(* CODESYS project CtaAppAbtauung_1.0.0.1.library
   Description: Abtauungs Library der CTA
   Version: 1.0.0.1
   Title: CtaAppAbtauung
   Author: SIS
   DocFormat: reStructuredText
   LanguageModelAttribute: qualified-access-only
   Placeholder: CtaAppAbtauung
   CompiledLibraryCompatibilityVersion: CODESYS V3.5 SP16 Patch 3
   Company: CTA
   DefaultNamespace: CtaAppAbtauung

Project tree, tasks and I/O mapping:
  libraries: CtaSysConfig, 1.0.0.2 (CTA); VisuSymbols, 4.5.0.0 (System); CtaVisSymbols, 1.0.0.1 (CTA); Standard, 3.5.18.0 (System); CtaAppInfluxLog, 1.0.0.1 (CTA); CtaVisApps, 1.0.0.0 (CTA); CtaVisHelp, 1.0.0.0 (CTA); CtaVisUser, 1.0.0.0 (CTA); WagoSysVisuBACnet, 2.0.0.0 (WAGO); WagoVisuIcons, 1.1.0.5 (WAGO); WagoVisuIconsMaterialDesign, 1.0.0.0 (WAGO); CtaAppBasic, 1.0.0.1 (CTA); CtaAppReport, 1.0.0.2 (CTA); CtaAppBmk, 1.0.0.0 (CTA); CtaAppTime, 1.0.0.1 (CTA)
  40 Visualizations/
    DIALOG/
      visualisation DIA_ParameterAbtauung
      visualisation DIA_Aussentemperatur
      visualisation DIA_Abtauukriterium
      visualisation DIA_Abtauuanforderung
    ICON/
      visualisation VIS_ABTAUUNG
      visualisation VIS_ABTAUUNG_CheckQuerry
      visualisation VIS_ABTAUUNG_OPEN
    visualisation VIS_AbtauungInfo
    visualisation VIS_AbtauungInfoQuerry
  30 Program Organization Units/
    function block fbAbtauung [ST]: actConfig, actTrendlog, actReport, actState, proAcknowledge, proAvailable, proLockDown, proIsError, proIsWarning, proConfigError, p_scAbtauungHilfsenergie_fbiRepTilLockdown, p_scAbtauungHilfsenergie_fbrTempAbtauEnde, p_scAbtauungHilfsenergie_fbtMaxAbtauungHiEnergie, p_scAbtauungHilfsenergie_fbudiAbtauungenHiEnergie, p_scAbtropfphase_fbtAbtropfzeit, p_scBase_fbtAbtauverzögerung, p_scBase_fbtSperrungAbtauung, p_scBase_fbrAtfürAbtauusperre, p_scManual_fbuiManualState, p_scManual_fbxManualResetLockTime, p_scUmluftabtauung_fbrTempAbtauUmluftOk, p_scUmluftabtauung_fbtAbtauzeitUmluft, p_scUmluftabtauung_fbudiAbtauungenUmluft, p_scAbtauukriterium_fbrAbtauukriteriumFix, p_scAbtauukriterium_fbrKorrekturAtLuftkühler, p_scTable_fbr_dT_Leistung1, p_scTable_fbr_dT_Leistung2, p_scTable_fbr_dT_LeistungMax, p_scTable_fbr_dT_LeistungMin, p_scTable_fbrAtLeistung1, p_scTable_fbrAtLeistung2, p_scTable_fbrAtLeistungMax, p_scTable_fbrAtLeistungMin, p_scTable_fbrAtMaxLeistung1, p_scTable_fbrAtMaxLeistung2, p_scTable_fbrAtMaxLeistungMax, p_scTable_fbrAtMaxLeistungMin, p_scTable_fbrAtMinLeistung1, p_scTable_fbrAtMinLeistung2, p_scTable_fbrAtMinLeistungMax, p_scTable_fbrAtMinLeistungMin, p_scTable_fbrAussenaemperaturMax, p_scTable_fbrAussentemperatur, p_scTable_fbrAussentemperaturMin, p_scTable_fbrLeistung1, p_scTable_fbrLeistung2, p_scTable_fbrMaxLeistung, p_scTable_fbrMinLeistung, p_scAussentemperatur_fbtAverageTimeRange, p_scAussentemperatur_fbxAtGemittelt, p_scInfluxDb_fbxEnable, proITF_REPORTMANAGER, prorActAussentemperatur, prorActAustrittstemperatur, prorZieltemperatur, prorActdTAbtauukriterium, prorAbtaukriteriumFix, prorKorrekturfaktorRk, prorActdTRückkühler, prordTAuslegung, prordTLeistung, proxSperrungAktiv, proudiActHilfsenergieAbtauungen, proudiActUmluftAbtaaungen, protSperrzeit, protStartverzögerung, proiStatus, proxAcknowledge, proxDemandAbtauung, proxDemandManualAbtauung, proxGenerelleDemand, proxDemandHilfsenergie, proManualUmluft, proManualHilfsenergie, proManualBeenden, proManualQuitTime, protTimeLeftAbtropfen, protTimeLeftUmluft, protTimeLeftHilfsenergie, protElapsedUmluft, protElapsedHilfsenergie
  00000000-0000-0000-0000-000000000000|D:\CoDeSys\LibrariesV3\trunk\Intern\CAA\CAA Template\3.4.0.0 draft\Placeholder.xml
  00000000-0000-0000-0000-000000000000|D:\CoDeSys\LibrariesV3\trunk\Intern\CAA\CAA Template\3.2.0.3 draft\Prefix.pdf
  00000000-0000-0000-0000-000000000000|D:\CoDeSys\LibrariesV3\trunk\Intern\CAA\CAA Template\3.5.2.0 draft\Placeholder.xml
  20 Structs/
    data type scParameter
    Abtauukriterium/
      Tabelle/
        data type scTable
      data type scAbtauukriterium
    Abtauuanforderung/
      data type scAbtauuanforderung
      Base/
        data type scBase
      Umluftabtauung/
        data type scUmluftabtauung
      AbtauungHilfsenergie/
        data type scAbtauungHilfsenergie
      Abtropfphase/
        data type scAbtropfphase
      Manual/
        data type scManual
    Aussentemperatur/
      data type scAussentemperatur
    Trend/
      data type scTrend
    InfluxDb/
      data type scInfluxDb
  50 Images/
  10 Documenation/
    global variables VersionHistory
    global variables readMe
  21 Interface/
    interface ITF_Abtauung: proAcknowledge, proAvailable, proLockDown, proIsError, proIsWarning, prorActdTAbtauukriterium, prorKorrekturfaktorRk, prorAbtaukriteriumFix, prorActAustrittstemperatur, prorActAussentemperatur, prorZieltemperatur, proxDemandAbtauung, proxDemandManualAbtauung, proxGenerelleDemand, proxDemandHilfsenergie, proxSperrungAktiv, proudiActUmluftAbtaaungen, proudiActHilfsenergieAbtauungen, protSperrzeit, protStartverzögerung, proiStatus, proxAcknowledge, prordTAuslegung, prordTLeistung, prorActdTRückkühler, protTimeLeftAbtropfen, protTimeLeftUmluft, protTimeLeftHilfsenergie, protElapsedUmluft, protElapsedHilfsenergie, p_scAbtauungHilfsenergie_fbudiAbtauungenHiEnergie, p_scAbtauungHilfsenergie_fbrTempAbtauEnde, p_scAbtauungHilfsenergie_fbtMaxAbtauungHiEnergie, p_scAbtauungHilfsenergie_fbiRepTilLockdown, p_scAbtropfphase_fbtAbtropfzeit, p_scBase_fbtAbtauverzögerung, p_scBase_fbtSperrungAbtauung, p_scBase_fbrAtfürAbtauusperre, p_scManual_fbxManualResetLockTime, p_scManual_fbuiManualState, p_scUmluftabtauung_fbrTempAbtauUmluftOk, p_scUmluftabtauung_fbtAbtauzeitUmluft, p_scUmluftabtauung_fbudiAbtauungenUmluft, p_scInfluxDb_fbxEnable, p_scAbtauukriterium_fbrAbtauukriteriumFix, p_scAbtauukriterium_fbrKorrekturAtLuftkühler, p_scTable_fbrAtLeistungMax, p_scTable_fbrAtMinLeistung1, p_scTable_fbr_dT_LeistungMin, p_scTable_fbrAtMaxLeistungMax, p_scTable_fbrAtMaxLeistung1, p_scTable_fbr_dT_Leistung2, p_scTable_fbr_dT_Leistung1, p_scTable_fbrAtMaxLeistung2, p_scTable_fbrAussenaemperaturMax, p_scTable_fbrAussentemperaturMin, p_scTable_fbrLeistung2, p_scTable_fbrMinLeistung, p_scTable_fbrAtMinLeistungMax, p_scTable_fbrAtLeistung1, p_scTable_fbrLeistung1, p_scTable_fbrMaxLeistung, p_scTable_fbrAussentemperatur, p_scTable_fbrAtMinLeistungMin, p_scTable_fbrAtMinLeistung2, p_scTable_fbrAtMaxLeistungMin, p_scTable_fbrAtLeistungMin, p_scTable_fbrAtLeistung2, p_scTable_fbr_dT_LeistungMax, p_scAussentemperatur_fbtAverageTimeRange, p_scAussentemperatur_fbxAtGemittelt, proConfigError, proITF_REPORTMANAGER, proManualUmluft, proManualHilfsenergie, proManualBeenden, proManualQuitTime
  11 Library Parameter/
  12 Konstanten/
  60 Textlisten/
    text list Error
    text list Info
    text list Warnung
  13 Globale Variablen/
    global variables GlobalKonstant
  text list GlobalTextList
*)

// 20 Structs/scParameter
TYPE scParameter :
    STRUCT
	// Parameter
	scAbtauuanforderung		:	scAbtauuanforderung;
	scAussentemperatur		:	scAussentemperatur;
	scAbtauukriterium		:	scAbtauukriterium;
	scInfluxDb				:	scInfluxDb;
	scTrend					:	scTrend;
    END_STRUCT
END_TYPE

// 20 Structs/Abtauukriterium/Tabelle/scTable
TYPE scTable :
	STRUCT
		(*Leistungen*)
		fbrMinLeistung				:	CtaSysConfig.fbREAL;
		fbrLeistung1				:	CtaSysConfig.fbREAL;
		fbrLeistung2				:	CtaSysConfig.fbREAL;
		fbrMaxLeistung				:	CtaSysConfig.fbREAL;
		(*Aussentemperaturen*)
		fbrAussentemperaturMin		:	CtaSysConfig.fbREAL;
		fbrAussentemperatur			:	CtaSysConfig.fbREAL;
		fbrAussenaemperaturMax		:	CtaSysConfig.fbREAL;
		(*dT*)
		fbrAtMinLeistungMin			:	CtaSysConfig.fbREAL;
		fbrAtMinLeistung1			:	CtaSysConfig.fbREAL;
		fbrAtMinLeistung2			:	CtaSysConfig.fbREAL;
		fbrAtMinLeistungMax			:	CtaSysConfig.fbREAL;		
		fbrAtLeistungMin			:	CtaSysConfig.fbREAL;
		fbrAtLeistung1				:	CtaSysConfig.fbREAL;
		fbrAtLeistung2				:	CtaSysConfig.fbREAL;
		fbrAtLeistungMax			:	CtaSysConfig.fbREAL;		
		fbrAtMaxLeistungMin			:	CtaSysConfig.fbREAL;
		fbrAtMaxLeistung1			:	CtaSysConfig.fbREAL;
		fbrAtMaxLeistung2			:	CtaSysConfig.fbREAL;
		fbrAtMaxLeistungMax			:	CtaSysConfig.fbREAL;
		(*dT's für Auslösungen*)
		fbr_dT_LeistungMin			:	CtaSysConfig.fbREAL;
		fbr_dT_Leistung1			:	CtaSysConfig.fbREAL;
		fbr_dT_Leistung2			:	CtaSysConfig.fbREAL;
		fbr_dT_LeistungMax			:	CtaSysConfig.fbREAL;
	END_STRUCT
END_TYPE

// 20 Structs/Abtauukriterium/scAbtauukriterium
TYPE scAbtauukriterium :
	STRUCT
		scTable 					:	scTable;
		fbrKorrekturAtLuftkühler	:	CtaSysConfig.fbREAL;		
		fbrAbtauukriteriumFix		:	CtaSysConfig.fbREAL;
	END_STRUCT
END_TYPE

// 20 Structs/Abtauuanforderung/scAbtauuanforderung
TYPE scAbtauuanforderung :
	STRUCT
		scBase					:	scBase;
		scUmluftabtauung		:	scUmluftabtauung;
		scAbtauungHilfsenergie	:	scAbtauungHilfsenergie;
		scAbtropfphase			:	scAbtropfphase;
		scManual				:	scManual;		
	END_STRUCT
END_TYPE

// 20 Structs/Aussentemperatur/scAussentemperatur
TYPE scAussentemperatur :
	STRUCT
		fbxAtGemittelt				:	CtaSysConfig.fbBOOL;
		fbtAverageTimeRange			:	CtaSysConfig.fbTIME;		
	END_STRUCT
END_TYPE

// 20 Structs/Abtauuanforderung/AbtauungHilfsenergie/scAbtauungHilfsenergie
TYPE scAbtauungHilfsenergie :
	STRUCT
		fbrTempAbtauEnde			:	CtaSysConfig.fbREAL;
		fbtMaxAbtauungHiEnergie		:	CtaSysConfig.fbTIME;
		fbiRepTilLockdown			:	CtaSysConfig.fbINT;
		fbudiAbtauungenHiEnergie	:	CtaSysConfig.fbUDINT;
	END_STRUCT
END_TYPE

// 20 Structs/Abtauuanforderung/Abtropfphase/scAbtropfphase
TYPE scAbtropfphase :
	STRUCT
		fbtAbtropfzeit				:	CtaSysConfig.fbTIME;	
	END_STRUCT
END_TYPE

// 20 Structs/Abtauuanforderung/Base/scBase
TYPE scBase :
	STRUCT
		fbtAbtauverzögerung			:	CtaSysConfig.fbTIME;
		fbtSperrungAbtauung			:	CtaSysConfig.fbTIME;
		fbrAtfürAbtauusperre		:	CtaSysConfig.fbREAL;
	END_STRUCT
END_TYPE

// 20 Structs/Abtauuanforderung/Manual/scManual
TYPE scManual :
	STRUCT
		fbxManualResetLockTime	:	CtaSysConfig.fbBOOL;	// Manuelle rücksetzung der Sperrzeit
		fbuiManualState			:	CtaSysConfig.fbUINT;	// 0 = Off, 1 = Umluftabtauung, 2 = Abtauung mit Hilfsenergie , 3 = Abtauung Beenden
	END_STRUCT
END_TYPE

// 20 Structs/Abtauuanforderung/Umluftabtauung/scUmluftabtauung
TYPE scUmluftabtauung :
	STRUCT
		fbrTempAbtauUmluftOk		:	CtaSysConfig.fbREAL;
		fbtAbtauzeitUmluft			:	CtaSysConfig.fbTIME;	
		fbudiAbtauungenUmluft		:	CtaSysConfig.fbUDINT;
	END_STRUCT
END_TYPE

// 20 Structs/Trend/scTrend
TYPE scTrend :
	STRUCT
		fbxEnable	: CtaSysConfig.fbBOOL;
	END_STRUCT
END_TYPE

// 20 Structs/InfluxDb/scInfluxDb
{attribute 'pack_mode' := '1'} 
TYPE scInfluxDb :
    STRUCT
        fbxEnable       :   CtaSysConfig.fbBOOL;
    END_STRUCT
END_TYPE

// 10 Documenation/VersionHistory
(* 

.. image:: ../../Images/CTA_Logo.jpg
   :align: right
   :width: 15% 

**Vorlage**   


============ =========== =========== ============================================
**Date**     **Version** **Author**  **Change**
------------ ----------- ----------- --------------------------------------------
04.03.2021   0.0.0.0     SIS         Vorlage erstellt

============ =========== =========== ============================================


*)
VAR_GLOBAL
    stInfo : STRING:= '0.0.0.0, Vorlage, CTA';
END_VAR

// 10 Documenation/readMe
(*

**ReadMe**
 
 |  **Empfehlung**
 |
 |	Bibliothek CtaAppPid zur implementierung eine PID- Reglers.
 |  Instanzieren Sie den CtaAppPid.fbPid in ihrem Funktionsbaustein oder POU beispielsweise als fbPidX(Komponente)Y. (X = Nr des Reglers; Komponente z.B Pumpe, Antrieb oder Ventilator; Y = Nr der Komponente) 
 |  Deklarieren Sie die Struktur Variable welche als Parameter und zur ansteuerung dienen wie im Code beispiel.
 |  
 |  *Beispiel* 

+-----------------------+---------------------------------------------------------------------------------------------------------------------------------------------------------------------------------------------------------------------------------------------------------------------------------------------------------------------------------------------------------------------------------------------------------------------------------------+
| Beschreibung          |  Code                                                                                                                                                                                                                                                                                                                                                                                                                                 |
+=======================+=======================================================================================================================================================================================================================================================================================================================================================================================================================================+
| Pou oder SmFb         | .. code-block:: codesys                                                                                                                                                                                                                                                                                                                                                                                                               |
|                       |                                                                                                                                                                                                                                                                                                                                                                                                                                       |
|                       |	// Deklaration als VAR im POU oder dem selbsterstellten Funktionsbaustein                                                                                                                                                                                                                                                                                                                                                       	|
|                       |   VAR   																																																																																																								|
|						|	    (*PID*)																																																	 																																																						|
|						|		fbPid1Pumpe1			: CtaAppPid.fbPid;                                                                                                                                                                                                                                                                                                                                                              						|
|                       | 		fbPid2Pumpe1			: CtaAppPid.fbPid;																																																																																														|
| 						|	END_VAR                                                                                                                                                                                                                                                                                                                                                                                                                         	|
+-----------------------+---------------------------------------------------------------------------------------------------------------------------------------------------------------------------------------------------------------------------------------------------------------------------------------------------------------------------------------------------------------------------------------------------------------------------------------+
| Code für Init         | .. code-block:: codesys                                                                                                                                                                                                                                                                                                                                                                                                               |
|                       |   																																																																																																									|
| 						|	// Kopieren des nachfolgenden Codes in eine Action zur Initialisierung der Parameter. Zum Beispiel actParameter.																																																																													|
|                       |	{region "Parameter Pid1Pumpe1"}                                                                                                                                                                                                                                                                                                                                                                                                     |
| 						|		(*Basis*)																																																																																																						|
|						|		fbPid1Pumpe1.scParameter.fbrDeadBand               		(_wertInit :=   0.0									, _minInit :=   	, _maxInit := 		);		//P1 Totband																																																														|
|						|		fbPid1Pumpe1.scParameter.fbrBand						(_wertInit :=   0.0									, _minInit :=   	, _maxInit := 		);		//P2 P- Band																																																														|
|						|		fbPid1Pumpe1.scParameter.fbrTn							(_wertInit :=   0.0									, _minInit :=   	, _maxInit := 		);		//P3 Nachstellzeit																																																													|
|						|		fbPid1Pumpe1.scParameter.fbrTv							(_wertInit :=   0.0									, _minInit :=   	, _maxInit := 		);		//P4 Vorhaltezeit																																																													|
|						|		fbPid1Pumpe1.scParameter.fbxInvert						(_wertInit := FALSE																			);		//P5 Regler Invertierung																																																											|
|						|	{endregion}                                                                                                                                                      																																																																	| 
+-----------------------+---------------------------------------------------------------------------------------------------------------------------------------------------------------------------------------------------------------------------------------------------------------------------------------------------------------------------------------------------------------------------------------------------------------------------------------+
*)                                                                                                                                                                                                                                                                                                                                                                                                                                                               
 VAR_GLOBAL                                                                                                                                                                                                                                                                                                                                                                                                                                                      
    xReadMeDone              :   BOOL;                                                                                                                                                                                                                                                                                                                                                                                                                           
END_VAR

// 13 Globale Variablen/GlobalKonstant
{attribute 'qualified_only'}
VAR_GLOBAL
	stReportTextListError   : CtaAppReport.stReportTextList := 'CtaAppAbtauung.Error';
	stReportTextListWarning : CtaAppReport.stReportTextList := 'CtaAppAbtauung.Warnung';
	stReportTextListInfo    : CtaAppReport.stReportTextList := 'CtaAppAbtauung.Info';	
END_VAR

// 30 Program Organization Units/fbAbtauung
FUNCTION_BLOCK fbAbtauung IMPLEMENTS ITF_Abtauung 
VAR_INPUT
	xRelease					:	BOOL;
	xAcknowledge				:	BOOL;
	xExtLockdown				:	BOOL;
	rActMaschienleistung		:	REAL;	
	rAussentemperatur			:	REAL;
	rAustrittstemperatur		:	REAL;	
	ITF_BMK						:	CtaAppBmk.ITF_BMK;
END_VAR
VAR_OUTPUT
	xDemandUmluft				:	BOOL;
	xDemandHilfsenergie			:	BOOL;
	xDemandAbtropfphase			:	BOOL;	
END_VAR
VAR
	(* Internal States *) 
	scEWI						:	CtaAppReport.scReportNr;
	_xIsWarning					:	BOOL;
	xIsWarning					:	BOOL;
	_xIsError					:	BOOL;
	xIsError					:	BOOL;
	xisEnabled					:	BOOL;

(* Hilfsvariablen *)
	rActdTAuslegung				:	REAL;
	rActdTLeistung				:	REAL;
	rAct_dT_Rückkühler			:	REAL;
	rAct_dT_Abtauukriterium		:	REAL;
	xAbtauen					:	BOOL;
	xAbtauungGestartet			:	BOOL;	
	rAussentemperaturGemittelt	:	REAL;
	xWasHilfsenergie			:	BOOL;
	xWasExternalLockdown		:	BOOL;
	
(* FB's *)
	// Skalierer		
	fbAbtauuScaler1				:	CtaAppBasic.fbscaleVierfach;
	fbAbtauuScaler2				:	CtaAppBasic.fbscaleVierfach;
	fbAbtauuScaler3				:	CtaAppBasic.fbscaleVierfach;	
	fbAbtauuScalerAuslegung		:	CtaAppBasic.fbscaleDreifach;	
	fbSclaerAbtauung			:	CtaAppBasic.fbscaleVierfach;
	// Gemittelte Aussentemperatur	
	fbAverageAt					:	CtaAppBasic.fbAverageAt;
		
(* Bistabile Sr *)
	srSperrungAbtauung			:	Standard.SR;
	
(* Flanken *)
	TRIG_SperrungAbtauung		:	Standard.F_TRIG;
	
(* Timer *)
	// Timer für Startverzögerung einer Abtauung
	TON_AbtauenDemand			:	Standard.TON;
	// Timer für Umluft abtauung	
	TON_AbtauungUmluft			:	Standard.TON;
	// Timer für Maximaldauer der Abtauung hilfsenergie
	TON_MaxAbtauung				:	Standard.TON;
	// Timer für Abtropfphase
	TON_Abtropfphase			:	Standard.TON;
	// Timer für Sperrung der nächsten Abtauung
	TON_SperrungAbtauung		:	Standard.TON;
	
(* Reports *)
	// Manager
	fbReportManager				:	CtaAppReport.fbReportManager;      
    // ForCounter
	difor						:	DINT;
	// Info Array's
	ayInfoReporter				:	ARRAY[1..2] OF CtaAppReport.fbReporter;
	// Info Abtauung mit Umluft gestartet
	xInfoAbtauungUmluft			:	BOOL;
	// Info Abtauung mit Hilfsenergie gestartet
	xInfoAbtauungHilfsenergie	:	BOOL;                                                            
	// Error Array's
	ayErrorReporter				:	ARRAY[1..2] OF CtaAppReport.fbReporter;
	// Error Abtauung zu lange gedauert
	xErrAbtauungToLong			:	BOOL;

(* Trendlogs *)
	fbTrendxAbtauanforderung	:	CtaAppInfluxLog.FB_LOG_NODE_BOOL;
	fbTrendxAbtauungGestartet	:	CtaAppInfluxLog.FB_LOG_NODE_BOOL;
	fbTrenddTAuslegung			:	CtaAppInfluxLog.FB_LOG_NODE_REAL;
	fbTrenddTLeistung			:	CtaAppInfluxLog.FB_LOG_NODE_REAL;
	fbAbtauukriterium			:	CtaAppInfluxLog.FB_LOG_NODE_REAL;
	fbTrendrdTRückkühler		:	CtaAppInfluxLog.FB_LOG_NODE_REAL;
	fbTrendxError				:	CtaAppInfluxLog.FB_LOG_NODE_BOOL;		
	
(* fbConfigfile *)
	fbConfigFile 				:	CtaSysConfig.fbConfigFile;
	xConfigError				:	BOOL;
	
(* Parameter *)
	scParameter					:	scParameter;
	
END_VAR

actConfig();

IF NOT xConfigError AND rAussentemperatur < scParameter.scAbtauuanforderung.scBase.fbrAtfürAbtauusperre.rValue THEN

	// Prüfen ob kürzlich eine Abtauung gestartet wurde
	TRIG_SperrungAbtauung(CLK	:=	(( xDemandUmluft OR xDemandHilfsenergie) AND xAcknowledge));
	
	// Abtauung sperren falls getriggert
	srSperrungAbtauung	(SET1	:=	TRIG_SperrungAbtauung.Q,
						 RESET	:= 	TON_SperrungAbtauung.Q	OR scParameter.scAbtauuanforderung.scManual.fbxManualResetLockTime.xValue );
						 
	IF scParameter.scAbtauuanforderung.scManual.fbxManualResetLockTime.xValue THEN
		scParameter.scAbtauuanforderung.scManual.fbxManualResetLockTime.proValue := FALSE;
	END_IF		
		 
	// Abtauung für dauer der Wiedereinschaltverzögerung sperren					
	TON_SperrungAbtauung	(IN		:=	srSperrungAbtauung.Q1,
						 	 PT		:=	scParameter.scAbtauuanforderung.scBase.fbtSperrungAbtauung.tValue);
						 
	// Prüfen der Fraigabe und Start der Abtauverzögerung bei Abtauuanforderung
	IF xRelease AND NOT srSperrungAbtauung.Q1 AND NOT xIsError THEN
		(* Scaler für die kleinste Aussentemperatur*)
		fbAbtauuScaler1			(rInput	:=	rActMaschienleistung		, 
								 x1		:=	scParameter.scAbtauukriterium.scTable.fbrMinLeistung.rValue				, 	// Kleinste Leistungsstufe
								 x2		:=	scParameter.scAbtauukriterium.scTable.fbrLeistung1.rValue				, 	// Mittlere Leistungsstufe 1
								 x3		:=	scParameter.scAbtauukriterium.scTable.fbrLeistung2.rValue				, 	// Mittlere Leistungsstufe 2
								 x4		:=	scParameter.scAbtauukriterium.scTable.fbrMaxLeistung.rValue				, 	// Grösste Leistungsstufe
								 y1		:=	scParameter.scAbtauukriterium.scTable.fbrAtMinLeistungMin.rValue		, 	// dT für kleinsete Leistungsstufe
								 y2		:=	scParameter.scAbtauukriterium.scTable.fbrAtMinLeistung1.rValue			, 	// dT für mittlere Leistungsstufe 1
								 y3		:=	scParameter.scAbtauukriterium.scTable.fbrAtMinLeistung2.rValue			, 	// dT für mittlere Leistungsstufe 2
								 y4		:=	scParameter.scAbtauukriterium.scTable.fbrAtMinLeistungMax.rValue		);	// dT für grösste Leistungsstufe
						
		(*Scaler für die mittlere Aussentemperatu*)	
		fbAbtauuScaler2			(rInput	:=	rActMaschienleistung		, 
								 x1		:=	scParameter.scAbtauukriterium.scTable.fbrMinLeistung.rValue				, 	// Kleinste Leistungsstufe         
								 x2		:=	scParameter.scAbtauukriterium.scTable.fbrLeistung1.rValue				, 	// Mittlere Leistungsstufe 1       
								 x3		:=	scParameter.scAbtauukriterium.scTable.fbrLeistung2.rValue				, 	// Mittlere Leistungsstufe 2       
								 x4		:=	scParameter.scAbtauukriterium.scTable.fbrMaxLeistung.rValue				, 	// Grösste Leistungsstufe          
								 y1		:=	scParameter.scAbtauukriterium.scTable.fbrAtLeistungMin.rValue			, 	// dT für kleinsete Leistungsstufe 
								 y2		:=	scParameter.scAbtauukriterium.scTable.fbrAtLeistung1.rValue				, 	// dT für mittlere Leistungsstufe 1
								 y3		:=	scParameter.scAbtauukriterium.scTable.fbrAtLeistung2.rValue				, 	// dT für mittlere Leistungsstufe 2
								 y4		:=	scParameter.scAbtauukriterium.scTable.fbrAtLeistungMax.rValue			);	// dT für grösste Leistungsstufe   
						 
		(*Scaler für die höchste Aussentemperatu*)
		fbAbtauuScaler3			(rInput	:=	rActMaschienleistung		, 
								 x1		:=	scParameter.scAbtauukriterium.scTable.fbrMinLeistung.rValue				, 	// Kleinste Leistungsstufe         
								 x2		:=	scParameter.scAbtauukriterium.scTable.fbrLeistung1.rValue				, 	// Mittlere Leistungsstufe 1       
								 x3		:=	scParameter.scAbtauukriterium.scTable.fbrLeistung2.rValue				, 	// Mittlere Leistungsstufe 2       
								 x4		:=	scParameter.scAbtauukriterium.scTable.fbrMaxLeistung.rValue				,	// Grösste Leistungsstufe          
								 y1		:=	scParameter.scAbtauukriterium.scTable.fbrAtMaxLeistungMin.rValue		, 	// dT für kleinsete Leistungsstufe 
								 y2		:=	scParameter.scAbtauukriterium.scTable.fbrAtMaxLeistung1.rValue			, 	// dT für mittlere Leistungsstufe 1
								 y3		:=	scParameter.scAbtauukriterium.scTable.fbrAtMaxLeistung2.rValue			, 	// dT für mittlere Leistungsstufe 2
								 y4		:=	scParameter.scAbtauukriterium.scTable.fbrAtMaxLeistungMax.rValue		);	// dT für grösste Leistungsstufe   
		
		(*Scaler für die Abtauung gemäss auslegung*)
		fbAbtauuScalerAuslegung	(rInput	:=	rAussentemperatur,
								 x1		:=	scParameter.scAbtauukriterium.scTable.fbrAussentemperaturMin.rValue		,	// kleinste Aussentemperatur
								 x2		:=	scParameter.scAbtauukriterium.scTable.fbrAussentemperatur.rValue		,	// mittlere Aussentemperatur
								 x3		:=	scParameter.scAbtauukriterium.scTable.fbrAussenaemperaturMax.rValue		,	// grösste Aussentemperatur
								 y1		:=	LIMIT(scParameter.scAbtauukriterium.scTable.fbrAtMinLeistungMin.rValue	,fbAbtauuScaler1.rOutput,	scParameter.scAbtauukriterium.scTable.fbrAtMinLeistungMax.rValue	),
								 y2		:=	LIMIT(scParameter.scAbtauukriterium.scTable.fbrAtLeistungMin.rValue		,fbAbtauuScaler2.rOutput,	scParameter.scAbtauukriterium.scTable.fbrAtLeistungMax.rValue		),
								 y3		:=	LIMIT(scParameter.scAbtauukriterium.scTable.fbrAtMaxLeistungMin.rValue	,fbAbtauuScaler2.rOutput,	scParameter.scAbtauukriterium.scTable.fbrAtMaxLeistungMax.rValue	));
		
		rActdTAuslegung := 	fbAbtauuScalerAuslegung.rOutput;
						
		(*Scaler für Abtauug gemäss Leistung*)
		fbSclaerAbtauung		(rInput	:=	rActMaschienleistung													, 
								 x1		:=	scParameter.scAbtauukriterium.scTable.fbrMinLeistung.rValue				, // Kleinste Leistungsstufe   
								 x2		:=	scParameter.scAbtauukriterium.scTable.fbrLeistung1.rValue				, // Mittlere Leistungsstufe 1 
								 x3		:=	scParameter.scAbtauukriterium.scTable.fbrLeistung2.rValue				, // Mittlere Leistungsstufe 2 
								 x4		:=	scParameter.scAbtauukriterium.scTable.fbrMaxLeistung.rValue				, // Grösste Leistungsstufe    
								 y1		:=	scParameter.scAbtauukriterium.scTable.fbr_dT_LeistungMin.rValue			, // dT für kleinsete Leistungsstufe 
								 y2		:=	scParameter.scAbtauukriterium.scTable.fbr_dT_Leistung1.rValue			, // dT für mittlere Leistungsstufe 1
								 y3		:=	scParameter.scAbtauukriterium.scTable.fbr_dT_Leistung2.rValue			, // dT für mittlere Leistungsstufe 2
								 y4		:=	scParameter.scAbtauukriterium.scTable.fbr_dT_LeistungMax.rValue			);// dT für grösste Leistungsstufe   
		
		rActdTLeistung	:=	LIMIT(scParameter.scAbtauukriterium.scTable.fbr_dT_LeistungMin.rValue,fbSclaerAbtauung.rOutput,scParameter.scAbtauukriterium.scTable.fbr_dT_LeistungMax.rValue);
					
		(*Berechnen und Festlegen des Abtaukriteriums*)	
		rAct_dT_Abtauukriterium := SEL	(scParameter.scAbtauukriterium.fbrAbtauukriteriumFix.rValue <> 0,
										 fbAbtauuScalerAuslegung.rOutput + LIMIT(scParameter.scAbtauukriterium.scTable.fbr_dT_LeistungMin.rValue,fbSclaerAbtauung.rOutput,scParameter.scAbtauukriterium.scTable.fbr_dT_LeistungMax.rValue)+scParameter.scAbtauukriterium.fbrKorrekturAtLuftkühler.rValue,
										 scParameter.scAbtauukriterium.fbrAbtauukriteriumFix.rValue) ;
		
		// Aussentemperatur mitteln						 
		fbAverageAt		(rAT := rAussentemperatur);								 
		rAussentemperaturGemittelt := fbAverageAt.GetAverageAT(TimeRange := scParameter.scAussentemperatur.fbtAverageTimeRange.proValue);	
										 
		(*Berechnung des aktuellen dT des Rückkühlers*)							 
		rAct_dT_Rückkühler := SEL(scParameter.scAussentemperatur.fbxAtGemittelt.xValue,rAussentemperatur,MIN(rAussentemperatur,rAussentemperaturGemittelt)) - rAustrittstemperatur;
		
		// Prüfen der Abtauuanforderung und Verzögern des Abtauustarts
		IF rAct_dT_Rückkühler >= rAct_dT_Abtauukriterium THEN
			TON_AbtauenDemand(IN	:=	TRUE									,
							 PT	:=	scParameter.scAbtauuanforderung.scBase.fbtAbtauverzögerung.tValue	,
							 Q	=>	xAbtauen								);
		ELSE
			TON_AbtauenDemand(IN	:= FALSE	);	
			xAbtauen				:= FALSE	 ;
		END_IF	
	ELSE
		TON_AbtauenDemand(IN	:= FALSE	);	
		xAbtauen	 			:= FALSE	 ;
		rAct_dT_Abtauukriterium	:= 0;
		rAct_dT_Rückkühler		:= 0;
	END_IF
	
	// Abtauuanforderung generieren
	IF NOT xIsError THEN
		// Starten einer manuellen Abtauung
		IF scParameter.scAbtauuanforderung.scManual.fbuiManualState.uiValue = 2 THEN
			xDemandHilfsenergie := TRUE;
			scParameter.scAbtauuanforderung.scManual.fbuiManualState.proValue := 0;
		ELSIF scParameter.scAbtauuanforderung.scManual.fbuiManualState.uiValue = 1 THEN
			xDemandUmluft		:= TRUE;
			scParameter.scAbtauuanforderung.scManual.fbuiManualState.proValue := 0;
		ELSE 
			// Starten einer Abtauung gemäss Abtauukriterium
			IF xAbtauen THEN
				IF rAussentemperatur > scParameter.scAbtauuanforderung.scUmluftabtauung.fbrTempAbtauUmluftOk.rValue THEN
					xDemandUmluft 		:= TRUE;
				ELSE	
					xDemandHilfsenergie := TRUE;
				END_IF		
			END_IF
		END_IF
	END_IF
	
	// Rückmeldung des Programms Abwarten um Timer zu starten
	IF xAcknowledge AND NOT xIsError THEN
		// Prüfen der geforderten Abtauung auf Umluft
		IF xDemandUmluft THEN
			TON_AbtauungUmluft(	IN	:= TRUE,
								PT	:= scParameter.scAbtauuanforderung.scUmluftabtauung.fbtAbtauzeitUmluft.tValue);
								
			IF NOT xAbtauungGestartet THEN				
				scParameter.scAbtauuanforderung.scUmluftabtauung.fbudiAbtauungenUmluft.proValue := scParameter.scAbtauuanforderung.scUmluftabtauung.fbudiAbtauungenUmluft.proValue + 1;
				xAbtauungGestartet := TRUE;
			END_IF	
			
			xInfoAbtauungUmluft		:= TRUE;
			
			IF TON_AbtauungUmluft.Q THEN
				xDemandUmluft 		:= FALSE;
				xAbtauungGestartet 	:= FALSE;
				xInfoAbtauungUmluft	:= FALSE;
			END_IF
			
		// Prüfen der geforderten Abtauung auf Hilfsenergie	
		ELSIF xDemandHilfsenergie THEN	
		
			IF NOT xAbtauungGestartet THEN				
				scParameter.scAbtauuanforderung.scAbtauungHilfsenergie.fbudiAbtauungenHiEnergie.proValue := scParameter.scAbtauuanforderung.scAbtauungHilfsenergie.fbudiAbtauungenHiEnergie.proValue + 1;
				xAbtauungGestartet := TRUE;
			END_IF	
			// Starten der Verzögerung
			TON_MaxAbtauung(IN := TRUE,
							PT := scParameter.scAbtauuanforderung.scAbtauungHilfsenergie.fbtMaxAbtauungHiEnergie.proValue);
				
			xInfoAbtauungHilfsenergie	:= TRUE;   
			xWasHilfsenergie			:= TRUE;
			
			// Wurde die Zieltemperatur erreicht wird Abtauung beendet
			IF 	rAustrittstemperatur >= scParameter.scAbtauuanforderung.scAbtauungHilfsenergie.fbrTempAbtauEnde.rValue THEN
				xDemandHilfsenergie			:= FALSE;
				xAbtauungGestartet  		:= FALSE;
				TON_MaxAbtauung			(IN	:= FALSE);
				xInfoAbtauungHilfsenergie	:= FALSE;
			// Zieltemperatur wird nicht innerhlab der eingestellten Frist erreicht = Error
			ELSIF TON_MaxAbtauung.Q THEN
				xErrAbtauungToLong			:= TRUE;
				xDemandHilfsenergie			:= FALSE;
				xAbtauungGestartet  		:= FALSE;
				TON_MaxAbtauung			(IN	:= FALSE);
				xInfoAbtauungHilfsenergie	:= FALSE;
			END_IF
			
		// Prüfen der geforderten Betriebsart auf Abtropfphase
		ELSIF xDemandAbtropfphase THEN
							
			// Starten der Verzögerung
			TON_Abtropfphase(	IN 	:= TRUE,
								PT 	:= scParameter.scAbtauuanforderung.scAbtropfphase.fbtAbtropfzeit.proValue);
								
			xWasHilfsenergie		:= FALSE;
					
			// Beenden der Abtropfphase						
			IF TON_Abtropfphase.Q THEN
				TON_Abtropfphase (IN	:= FALSE);							
				xDemandAbtropfphase		:= FALSE;	
			END_IF
					
		ELSE
			TON_AbtauungUmluft	(IN	:= FALSE);
			TON_MaxAbtauung		(IN := FALSE);
			TON_Abtropfphase	(IN	:= FALSE);
		END_IF
	ELSIF NOT xAcknowledge AND NOT xIsError THEN
		IF xWasExternalLockdown THEN
			// Zurücketzen der Timer wenn Lockdown von Ausserhalb des FB's kommt.
			TON_AbtauungUmluft	(IN	:= FALSE);
			TON_MaxAbtauung		(IN := FALSE);
			TON_Abtropfphase	(IN	:= FALSE);
			xWasExternalLockdown	:= FALSE;
		ELSE
			IF xWasHilfsenergie THEN
				xDemandAbtropfphase := TRUE;
			END_IF
		END_IF
		
	ELSIF NOT xAcknowledge AND xIsError THEN
		// Auslösung von xIsError durch Abtauung Hilfsenergie - Wurde nicht innerhalb der Frist erricht
		IF  xIsError THEN
			TON_AbtauungUmluft	(IN	:= FALSE);
			TON_MaxAbtauung		(IN := FALSE);
			TON_Abtropfphase	(IN	:= FALSE);			
			xDemandUmluft			:= FALSE;
			xDemandHilfsenergie		:= FALSE;
			xDemandAbtropfphase		:= TRUE;	// Entsprechend wird Abtropfphase nach wie vor angefordert.
			xErrAbtauungToLong		:= FALSE;	// Zurücksetzen des Fehlers
		END_IF
	END_IF
	
	IF scParameter.scAbtauuanforderung.scManual.fbuiManualState.uiValue = 3 THEN
		// Infos zurücksetzen 
		xInfoAbtauungUmluft			:= FALSE;
		xInfoAbtauungHilfsenergie	:= FALSE;
		// Error zurücksetzen
		xErrAbtauungToLong			:= FALSE;
		// Timer Zurücksetzen
		TON_AbtauungUmluft		(IN	:= FALSE);
		TON_MaxAbtauung			(IN := FALSE);
		TON_Abtropfphase		(IN	:= FALSE);
		// Demands zurücksetzen
		xDemandUmluft				:= FALSE;
		xDemandHilfsenergie			:= FALSE;
		xDemandAbtropfphase			:= FALSE;
		xWasExternalLockdown		:= FALSE;
		// Manualstate zurücksetzen
		IF NOT xAcknowledge THEN
			scParameter.scAbtauuanforderung.scManual.fbuiManualState.proValue := 0;
		END_IF
	END_IF	
	
	IF xExtLockdown AND NOT xIsError THEN
		xWasExternalLockdown	:= TRUE;
	END_IF
	
	// Reports
	IF __QUERYINTERFACE(ITF_BMK,ITF_BMK)THEN
		actReport();
	END_IF
ELSE // Im falle eines Configerrors wird alles zurückgesetzt
	xDemandUmluft				:= FALSE;
	xDemandHilfsenergie 		:= FALSE;
	xDemandAbtropfphase			:= FALSE;
	xInfoAbtauungUmluft			:= FALSE;
	xInfoAbtauungHilfsenergie	:= FALSE;
	xErrAbtauungToLong			:= FALSE;
	TON_AbtauungUmluft		(IN	:= FALSE);
	TON_MaxAbtauung			(IN := FALSE);
	TON_Abtropfphase		(IN	:= FALSE);
	xWasExternalLockdown		:= FALSE;
	
	// Konfigurationsfehler
	IF xConfigError THEN
		IF __QUERYINTERFACE(ITF_BMK,ITF_BMK)THEN
			actReport();
		END_IF
	END_IF
END_IF

// Status
actState();

// Trends
IF __QUERYINTERFACE(ITF_BMK,ITF_BMK) THEN
	actTrendlog();
END_IF

ACTION actConfig:
fbConfigFile();

(*ABTAUANFORDERUNG*)
	(*Base*)
	scParameter.scAbtauuanforderung.scBase.fbtAbtauverzögerung						(_usiParaNr :=  1,	itfConfigFb := fbConfigFile, _WertInit:= T#10M, _MinInit := T#00M,_MaxInit := T#60M	);
	scParameter.scAbtauuanforderung.scBase.fbtSperrungAbtauung						(_usiParaNr :=  2,	itfConfigFb := fbConfigFile, _WertInit:= T#30M, _MinInit := T#00M,_MaxInit := T#24H	);
	(*Umluftabtauung*)
	scParameter.scAbtauuanforderung.scUmluftabtauung.fbrTempAbtauUmluftOk			(_usiParaNr :=  3,	itfConfigFb := fbConfigFile, _WertInit:= 12.00, _MinInit := -50.0,_MaxInit :=  50.0	);
	scParameter.scAbtauuanforderung.scUmluftabtauung.fbtAbtauzeitUmluft				(_usiParaNr :=  4,	itfConfigFb := fbConfigFile, _WertInit:= T#30M, _MinInit := T#00M,_MaxInit := T#24H	);
	scParameter.scAbtauuanforderung.scUmluftabtauung.fbudiAbtauungenUmluft			(_usiParaNr :=  5,	itfConfigFb := fbConfigFile, _WertInit:= 00000, 									);
	(*Abtauung Hilfsenergie*)
	scParameter.scAbtauuanforderung.scAbtauungHilfsenergie.fbrTempAbtauEnde			(_usiParaNr :=  6,	itfConfigFb := fbConfigFile, _WertInit:= 10.00, _MinInit := -50.0,_MaxInit :=  50.0	);
	scParameter.scAbtauuanforderung.scAbtauungHilfsenergie.fbtMaxAbtauungHiEnergie	(_usiParaNr :=  7,	itfConfigFb := fbConfigFile, _WertInit:= T#10M, _MinInit := T#00M,_MaxInit := T#24H	);
	scParameter.scAbtauuanforderung.scAbtauungHilfsenergie.fbiRepTilLockdown		(_usiParaNr :=  8,	itfConfigFb := fbConfigFile, _WertInit:= 00003, 									);
	scParameter.scAbtauuanforderung.scAbtauungHilfsenergie.fbudiAbtauungenHiEnergie	(_usiParaNr :=  9,	itfConfigFb := fbConfigFile, _WertInit:= 00000, 									);
	(*Abtropfphase*)
	scParameter.scAbtauuanforderung.scAbtropfphase.fbtAbtropfzeit					(_usiParaNr := 10,	itfConfigFb := fbConfigFile, _WertInit:= T#10M, _MinInit := T#00M,_MaxInit := T#24H	);
	(*Manuell*)
	scParameter.scAbtauuanforderung.scManual.fbuiManualState						(_usiParaNr := 11,	itfConfigFb := fbConfigFile, _WertInit:= 00000, _MinInit := 00000,_MaxInit := 00003	);
(*ABTAUUKRITERIUM*)	
	(*TABLE*)
		(*Tabele Vertikal*)
		scParameter.scAbtauukriterium.scTable.fbrMinLeistung			(_usiParaNr := 12,	itfConfigFb := fbConfigFile, _MinInit :=   0.0,_MaxInit := 100.0);
		scParameter.scAbtauukriterium.scTable.fbrLeistung1				(_usiParaNr := 13,	itfConfigFb := fbConfigFile, _MinInit :=   0.0,_MaxInit := 100.0);
		scParameter.scAbtauukriterium.scTable.fbrLeistung2				(_usiParaNr := 14,	itfConfigFb := fbConfigFile, _MinInit :=   0.0,_MaxInit := 100.0);
		scParameter.scAbtauukriterium.scTable.fbrMaxLeistung			(_usiParaNr := 15,	itfConfigFb := fbConfigFile, _MinInit :=   0.0,_MaxInit := 100.0);
		(*Tabelle Horizontal*)
		scParameter.scAbtauukriterium.scTable.fbrAussentemperaturMin	(_usiParaNr := 16,	itfConfigFb := fbConfigFile, _MinInit := -50.0,_MaxInit :=  50.0);
		scParameter.scAbtauukriterium.scTable.fbrAussentemperatur		(_usiParaNr := 17,	itfConfigFb := fbConfigFile, _MinInit := -50.0,_MaxInit :=  50.0);
		scParameter.scAbtauukriterium.scTable.fbrAussenaemperaturMax	(_usiParaNr := 18,	itfConfigFb := fbConfigFile, _MinInit := -50.0,_MaxInit :=  50.0);
		(*Tabellen Daten*)
		scParameter.scAbtauukriterium.scTable.fbrAtMinLeistungMin		(_usiParaNr := 19,	itfConfigFb := fbConfigFile, _MinInit := -50.0,_MaxInit :=  50.0);
		scParameter.scAbtauukriterium.scTable.fbrAtMinLeistung1			(_usiParaNr := 20,	itfConfigFb := fbConfigFile, _MinInit := -50.0,_MaxInit :=  50.0);
		scParameter.scAbtauukriterium.scTable.fbrAtMinLeistung2			(_usiParaNr := 21,	itfConfigFb := fbConfigFile, _MinInit := -50.0,_MaxInit :=  50.0);
		scParameter.scAbtauukriterium.scTable.fbrAtMinLeistungMax		(_usiParaNr := 22,	itfConfigFb := fbConfigFile, _MinInit := -50.0,_MaxInit :=  50.0);
		scParameter.scAbtauukriterium.scTable.fbrAtLeistungMin			(_usiParaNr := 23,	itfConfigFb := fbConfigFile, _MinInit := -50.0,_MaxInit :=  50.0);
		scParameter.scAbtauukriterium.scTable.fbrAtLeistung1			(_usiParaNr := 24,	itfConfigFb := fbConfigFile, _MinInit := -50.0,_MaxInit :=  50.0);
		scParameter.scAbtauukriterium.scTable.fbrAtLeistung2			(_usiParaNr := 25,	itfConfigFb := fbConfigFile, _MinInit := -50.0,_MaxInit :=  50.0);
		scParameter.scAbtauukriterium.scTable.fbrAtLeistungMax			(_usiParaNr := 26,	itfConfigFb := fbConfigFile, _MinInit := -50.0,_MaxInit :=  50.0);
		scParameter.scAbtauukriterium.scTable.fbrAtMaxLeistungMin		(_usiParaNr := 27,	itfConfigFb := fbConfigFile, _MinInit := -50.0,_MaxInit :=  50.0);
		scParameter.scAbtauukriterium.scTable.fbrAtMaxLeistung1			(_usiParaNr := 28,	itfConfigFb := fbConfigFile, _MinInit := -50.0,_MaxInit :=  50.0);
		scParameter.scAbtauukriterium.scTable.fbrAtMaxLeistung2			(_usiParaNr := 29,	itfConfigFb := fbConfigFile, _MinInit := -50.0,_MaxInit :=  50.0);
		scParameter.scAbtauukriterium.scTable.fbrAtMaxLeistungMax		(_usiParaNr := 30,	itfConfigFb := fbConfigFile, _MinInit := -50.0,_MaxInit :=  50.0);
		(*dT Auslösungen*)
		scParameter.scAbtauukriterium.scTable.fbr_dT_LeistungMin		(_usiParaNr := 31,	itfConfigFb := fbConfigFile, _MinInit :=   0.0,_MaxInit :=  20.0);
		scParameter.scAbtauukriterium.scTable.fbr_dT_Leistung1			(_usiParaNr := 32,	itfConfigFb := fbConfigFile, _MinInit :=   0.0,_MaxInit :=  20.0);
		scParameter.scAbtauukriterium.scTable.fbr_dT_Leistung2			(_usiParaNr := 33,	itfConfigFb := fbConfigFile, _MinInit :=   0.0,_MaxInit :=  20.0);
		scParameter.scAbtauukriterium.scTable.fbr_dT_LeistungMax		(_usiParaNr := 34,	itfConfigFb := fbConfigFile, _MinInit :=   0.0,_MaxInit :=  20.0);
	(* Sonstige *)
	scParameter.scAbtauukriterium.fbrKorrekturAtLuftkühler				(_usiParaNr := 35,	itfConfigFb := fbConfigFile, _MinInit := -20.0,_MaxInit :=  20.0);
	scParameter.scAbtauukriterium.fbrAbtauukriteriumFix					(_usiParaNr := 36,	itfConfigFb := fbConfigFile, _MinInit := -20.0,_MaxInit :=  20.0);
(*AUSSENTEMPERATUR*)
	scParameter.scAussentemperatur.fbxAtGemittelt						(_usiParaNr := 37,	itfConfigFb := fbConfigFile, _WertInit:= FALSE, 									);
	scParameter.scAussentemperatur.fbtAverageTimeRange					(_usiParaNr := 38,	itfConfigFb := fbConfigFile, _WertInit:= T#24H, _MinInit := T#00M,_MaxInit := T#7D	);
(*Influx DB*)
	scParameter.scInfluxDb.fbxEnable									(_usiParaNr := 39,	itfConfigFb := fbConfigFile, _WertInit:=  TRUE, 									);													
(*Trendaufzeichnung*)
	scParameter.scTrend.fbxEnable										(_usiParaNr := 40,	itfConfigFb := fbConfigFile, _WertInit:=  TRUE, 									);
(* Abtausperrung*)	
scParameter.scAbtauuanforderung.scBase.fbrAtfürAbtauusperre				(_usiParaNr := 41,	itfConfigFb := fbConfigFile, _WertInit:= 15.00, _MinInit := -50.0,_MaxInit :=  50.0	);
END_ACTION

ACTION actTrendlog:
(* Abtauuanforderung *)
fbTrendxAbtauanforderung.ENABLE		:=	scParameter.scTrend.fbxEnable.proValue AND
										scParameter.scInfluxDb.fbxEnable.proValue;
fbTrendxAbtauanforderung.KEY		:=	CONCAT(ITF_BMK.proGetObjectId,'_Abtauuanforderung');
fbTrendxAbtauanforderung.SET_VALUE	:=	xAbtauen;

(* Abtauung gestartet *)
fbTrendxAbtauungGestartet.ENABLE	:=	scParameter.scTrend.fbxEnable.proValue AND
										scParameter.scInfluxDb.fbxEnable.proValue;
fbTrendxAbtauungGestartet.KEY		:=	CONCAT(ITF_BMK.proGetObjectId,'_Abtauung_gestartet');
fbTrendxAbtauungGestartet.SET_VALUE	:=  xAbtauungGestartet;

(* dT aus der Auslegung *)
fbTrenddTAuslegung.ENABLE			:=	scParameter.scTrend.fbxEnable.proValue AND
										scParameter.scInfluxDb.fbxEnable.proValue;
fbTrenddTAuslegung.KEY				:=	CONCAT(ITF_BMK.proGetObjectId,'_dT_Auslegung');
fbTrenddTAuslegung.SET_VALUE		:=  rActdTAuslegung;

(* dT aus der Maschinenleistung *)
fbTrenddTLeistung.ENABLE			:=	scParameter.scTrend.fbxEnable.proValue AND
										scParameter.scInfluxDb.fbxEnable.proValue;
fbTrenddTLeistung.KEY 				:=	CONCAT(ITF_BMK.proGetObjectId,'_dT_Leistung');
fbTrenddTLeistung.SET_VALUE			:=  rActdTLeistung;

(* Abtauukriterium aus Auslegung und Leistung *)
fbAbtauukriterium.ENABLE			:=	scParameter.scTrend.fbxEnable.proValue AND
										scParameter.scInfluxDb.fbxEnable.proValue;
fbAbtauukriterium.KEY 				:=	CONCAT(ITF_BMK.proGetObjectId,'_dT_Abtauukriterium');
fbAbtauukriterium.SET_VALUE			:=  rAct_dT_Abtauukriterium;

(* dT des Rückkühlers At zu Austritt *)
fbTrendrdTRückkühler.ENABLE			:=	scParameter.scTrend.fbxEnable.proValue AND
										scParameter.scInfluxDb.fbxEnable.proValue;
fbTrendrdTRückkühler.KEY 			:=	CONCAT(ITF_BMK.proGetObjectId,'_dT_Rückkühler');
fbTrendrdTRückkühler.SET_VALUE		:=  rAct_dT_Rückkühler;

(* Fehler *)
fbTrendxError.ENABLE				:=	scParameter.scTrend.fbxEnable.proValue AND
										scParameter.scInfluxDb.fbxEnable.proValue;
fbTrendxError.KEY 					:=	CONCAT(ITF_BMK.proGetObjectId,'_Abtauung_xError');
fbTrendxError.SET_VALUE				:=  xIsError;
END_ACTION

ACTION actReport:
(* EWI Manager *)
fbReportManager(	stErrorInitReportTextListIn		:=	ADR(GlobalKonstant.stReportTextListError),
					stWarningInitReportTextListIn	:=	ADR(GlobalKonstant.stReportTextListWarning),
					stInfoInitReportTextListIn		:=	ADR(GlobalKonstant.stReportTextListInfo),
					scReportNr						:=	scEWI);
					
(* Errors *)                        
        (* Meldung Error Abtauung zu lange gedauert *)
        ayErrorReporter[1].proPrio  := 2;
        ayErrorReporter[1].metReport(     		xSetReportIn					:= xErrAbtauungToLong,
												iReportID						:= 1,
												enReportTypeIn					:= CtaAppReport.enReportType.Error,  
												enReportAcknowledgeTypeIn   	:= CtaAppReport.enReportacknowledgeType.RetryN,
												tDelay							:= T#0S, 
												ITF_BMK_IN						:= ITF_BMK,			              
												pstReportTextListIn				:= ADR(GlobalKonstant.stReportTextListError),
												stOptionalReportText		    := '',   
												iRetryTilReportLock 		    := scParameter.scAbtauuanforderung.scAbtauungHilfsenergie.fbiRepTilLockdown.iValue, 
												xResetCount         		    := FALSE,  
												tReset						    := T#24H); 
								
		(* Meldung Configerror *)
        ayErrorReporter[2].proPrio  := 1;
        ayErrorReporter[2].metReport(     		xSetReportIn					:= xConfigError,
												iReportID						:= 2,
												enReportTypeIn					:= CtaAppReport.enReportType.Error,  
												enReportAcknowledgeTypeIn   	:= CtaAppReport.enReportacknowledgeType.Quit,
												tDelay							:= T#0S, 
												ITF_BMK_IN						:= ITF_BMK,			              
												pstReportTextListIn				:= ADR(GlobalKonstant.stReportTextListError),
												stOptionalReportText		    := '',   
												iRetryTilReportLock 		    := 0, 
												xResetCount         		    := FALSE,  
												tReset						    := T#24H);
	
(* Infos *)      
        (* Info Abtauung Umluft gestartet *)      
        ayInfoReporter[1].proPrio := 2;
        ayInfoReporter[1].metReport(			xSetReportIn					:= xInfoAbtauungUmluft AND xAcknowledge,
												iReportID						:= 1,
												enReportTypeIn					:= CtaAppReport.enReportType.Info,  
												enReportAcknowledgeTypeIn   	:= CtaAppReport.enReportAcknowledgeType.Auto,
												tDelay							:= T#0S, 
												ITF_BMK_IN						:= ITF_BMK,			              
												pstReportTextListIn				:= ADR(GlobalKonstant.stReportTextListInfo),
												stOptionalReportText		    := '',   
												iRetryTilReportLock 		    := 0, 
												xResetCount         		    := FALSE,  
												tReset						    := T#24H);  
												
		(* Info Abtauung Hilfsenergie gestartet *)      
        ayInfoReporter[2].proPrio := 2;
        ayInfoReporter[2].metReport(			xSetReportIn					:= xInfoAbtauungHilfsenergie AND xAcknowledge ,
												iReportID						:= 2,
												enReportTypeIn					:= CtaAppReport.enReportType.Info,  
												enReportAcknowledgeTypeIn   	:= CtaAppReport.enReportAcknowledgeType.Auto,
												tDelay							:= T#0S, 
												ITF_BMK_IN						:= ITF_BMK,			              
												pstReportTextListIn				:= ADR(GlobalKonstant.stReportTextListInfo),
												stOptionalReportText		    := '',   
												iRetryTilReportLock 		    := 0, 
												xResetCount         		    := FALSE,  
												tReset						    := T#24H);            
												
(* Sync Reports *)                                         
FOR difor := LOWER_BOUND(ayErrorReporter,1) TO UPPER_BOUND(ayErrorReporter,1) DO
	fbReportManager.metSyncReporter(ayErrorReporter[difor]);	
END_FOR;
FOR difor := LOWER_BOUND(ayInfoReporter,1) TO UPPER_BOUND(ayInfoReporter,1) DO
	fbReportManager.metSyncReporter(ayInfoReporter[difor]);	
END_FOR;
                                                                             
_xIsError   := scEWI.iError <> 0;
_xIsWarning := scEWI.iWarning <> 0;
END_ACTION

ACTION actState:
xisEnabled  :=  NOT xConfigError;
xIsWarning 	:= _xIsWarning;
xIsError	:= _xIsError;
END_ACTION

{attribute 'monitoring' := 'variable'}
PROPERTY proAcknowledge : BOOL
GET
proAcknowledge := NOT proIsError;
END_GET
END_PROPERTY

{attribute 'monitoring' := 'variable'}
PROPERTY proAvailable : BOOL
GET
proAvailable := NOT proIsError;
END_GET
END_PROPERTY

{attribute 'monitoring' := 'variable'}
PROPERTY proLockDown : BOOL
GET
proLockDown := proIsError;
END_GET
END_PROPERTY

PROPERTY proIsError : BOOL
GET
proIsError := xIsError;
END_GET
END_PROPERTY

PROPERTY proIsWarning : BOOL
GET
proIsWarning := xIsWarning;
END_GET
END_PROPERTY

PROPERTY proConfigError : BOOL
GET
proConfigError := xConfigError;
END_GET
END_PROPERTY

PROPERTY p_scAbtauungHilfsenergie_fbiRepTilLockdown : CtaSysConfig.ITF_DATATYPE
GET
p_scAbtauungHilfsenergie_fbiRepTilLockdown := scParameter.scAbtauuanforderung.scAbtauungHilfsenergie.fbiRepTilLockdown;
END_GET
END_PROPERTY

PROPERTY p_scAbtauungHilfsenergie_fbrTempAbtauEnde : CtaSysConfig.ITF_DATATYPE
GET
p_scAbtauungHilfsenergie_fbrTempAbtauEnde := scParameter.scAbtauuanforderung.scAbtauungHilfsenergie.fbrTempAbtauEnde;
END_GET
END_PROPERTY

PROPERTY p_scAbtauungHilfsenergie_fbtMaxAbtauungHiEnergie : CtaSysConfig.ITF_DATATYPE
GET
p_scAbtauungHilfsenergie_fbtMaxAbtauungHiEnergie := scParameter.scAbtauuanforderung.scAbtauungHilfsenergie.fbtMaxAbtauungHiEnergie;
END_GET
END_PROPERTY

PROPERTY p_scAbtauungHilfsenergie_fbudiAbtauungenHiEnergie : CtaSysConfig.ITF_DATATYPE
GET
p_scAbtauungHilfsenergie_fbudiAbtauungenHiEnergie := scParameter.scAbtauuanforderung.scAbtauungHilfsenergie.fbudiAbtauungenHiEnergie;
END_GET
END_PROPERTY

PROPERTY p_scAbtropfphase_fbtAbtropfzeit : CtaSysConfig.ITF_DATATYPE
GET
p_scAbtropfphase_fbtAbtropfzeit := scParameter.scAbtauuanforderung.scAbtropfphase.fbtAbtropfzeit;
END_GET
END_PROPERTY

PROPERTY p_scBase_fbtAbtauverzögerung : CtaSysConfig.ITF_DATATYPE
GET
p_scBase_fbtAbtauverzögerung := scParameter.scAbtauuanforderung.scBase.fbtAbtauverzögerung;
END_GET
END_PROPERTY

PROPERTY p_scBase_fbtSperrungAbtauung : CtaSysConfig.ITF_DATATYPE
GET
p_scBase_fbtSperrungAbtauung := scParameter.scAbtauuanforderung.scBase.fbtSperrungAbtauung;
END_GET
END_PROPERTY

PROPERTY p_scBase_fbrAtfürAbtauusperre : CtaSysConfig.ITF_DATATYPE
GET
p_scBase_fbrAtfürAbtauusperre := scParameter.scAbtauuanforderung.scBase.fbrAtfürAbtauusperre;
END_GET
END_PROPERTY

PROPERTY p_scManual_fbuiManualState : CtaSysConfig.ITF_DATATYPE
GET
p_scManual_fbuiManualState := scParameter.scAbtauuanforderung.scManual.fbuiManualState;
END_GET
END_PROPERTY

PROPERTY p_scManual_fbxManualResetLockTime : CtaSysConfig.ITF_DATATYPE
GET
p_scManual_fbxManualResetLockTime := scParameter.scAbtauuanforderung.scManual.fbxManualResetLockTime;
END_GET
END_PROPERTY

PROPERTY p_scUmluftabtauung_fbrTempAbtauUmluftOk : CtaSysConfig.ITF_DATATYPE
GET
p_scUmluftabtauung_fbrTempAbtauUmluftOk := scParameter.scAbtauuanforderung.scUmluftabtauung.fbrTempAbtauUmluftOk;
END_GET
END_PROPERTY

PROPERTY p_scUmluftabtauung_fbtAbtauzeitUmluft : CtaSysConfig.ITF_DATATYPE
GET
p_scUmluftabtauung_fbtAbtauzeitUmluft := scParameter.scAbtauuanforderung.scUmluftabtauung.fbtAbtauzeitUmluft;
END_GET
END_PROPERTY

PROPERTY p_scUmluftabtauung_fbudiAbtauungenUmluft : CtaSysConfig.ITF_DATATYPE
GET
p_scUmluftabtauung_fbudiAbtauungenUmluft := scParameter.scAbtauuanforderung.scUmluftabtauung.fbudiAbtauungenUmluft;
END_GET
END_PROPERTY

PROPERTY p_scAbtauukriterium_fbrAbtauukriteriumFix : CtaSysConfig.ITF_DATATYPE
GET
p_scAbtauukriterium_fbrAbtauukriteriumFix := scParameter.scAbtauukriterium.fbrAbtauukriteriumFix;
END_GET
END_PROPERTY

PROPERTY p_scAbtauukriterium_fbrKorrekturAtLuftkühler : CtaSysConfig.ITF_DATATYPE
GET
p_scAbtauukriterium_fbrKorrekturAtLuftkühler := scParameter.scAbtauukriterium.fbrKorrekturAtLuftkühler;
END_GET
END_PROPERTY

PROPERTY p_scTable_fbr_dT_Leistung1 : CtaSysConfig.ITF_DATATYPE
GET
p_scTable_fbr_dT_Leistung1 := scParameter.scAbtauukriterium.scTable.fbr_dT_Leistung1;
END_GET
END_PROPERTY

PROPERTY p_scTable_fbr_dT_Leistung2 : CtaSysConfig.ITF_DATATYPE
GET
p_scTable_fbr_dT_Leistung2 := scParameter.scAbtauukriterium.scTable.fbr_dT_Leistung2;
END_GET
END_PROPERTY

PROPERTY p_scTable_fbr_dT_LeistungMax : CtaSysConfig.ITF_DATATYPE
GET
p_scTable_fbr_dT_LeistungMax := scParameter.scAbtauukriterium.scTable.fbr_dT_LeistungMax;
END_GET
END_PROPERTY

PROPERTY p_scTable_fbr_dT_LeistungMin : CtaSysConfig.ITF_DATATYPE
GET
p_scTable_fbr_dT_LeistungMin := scParameter.scAbtauukriterium.scTable.fbr_dT_LeistungMin;
END_GET
END_PROPERTY

PROPERTY p_scTable_fbrAtLeistung1 : CtaSysConfig.ITF_DATATYPE
GET
p_scTable_fbrAtLeistung1 := scParameter.scAbtauukriterium.scTable.fbrAtLeistung1;
END_GET
END_PROPERTY

PROPERTY p_scTable_fbrAtLeistung2 : CtaSysConfig.ITF_DATATYPE
GET
p_scTable_fbrAtLeistung2 := scParameter.scAbtauukriterium.scTable.fbrAtLeistung2;
END_GET
END_PROPERTY

PROPERTY p_scTable_fbrAtLeistungMax : CtaSysConfig.ITF_DATATYPE
GET
p_scTable_fbrAtLeistungMax := scParameter.scAbtauukriterium.scTable.fbrAtLeistungMax;
END_GET
END_PROPERTY

PROPERTY p_scTable_fbrAtLeistungMin : CtaSysConfig.ITF_DATATYPE
GET
p_scTable_fbrAtLeistungMin := scParameter.scAbtauukriterium.scTable.fbrAtLeistungMin;
END_GET
END_PROPERTY

PROPERTY p_scTable_fbrAtMaxLeistung1 : CtaSysConfig.ITF_DATATYPE
GET
p_scTable_fbrAtMaxLeistung1 := scParameter.scAbtauukriterium.scTable.fbrAtMaxLeistung1;
END_GET
END_PROPERTY

PROPERTY p_scTable_fbrAtMaxLeistung2 : CtaSysConfig.ITF_DATATYPE
GET
p_scTable_fbrAtMaxLeistung2 := scParameter.scAbtauukriterium.scTable.fbrAtMaxLeistung2;
END_GET
END_PROPERTY

PROPERTY p_scTable_fbrAtMaxLeistungMax : CtaSysConfig.ITF_DATATYPE
GET
p_scTable_fbrAtMaxLeistungMax := scParameter.scAbtauukriterium.scTable.fbrAtMaxLeistungMax;
END_GET
END_PROPERTY

PROPERTY p_scTable_fbrAtMaxLeistungMin : CtaSysConfig.ITF_DATATYPE
GET
p_scTable_fbrAtMaxLeistungMin := scParameter.scAbtauukriterium.scTable.fbrAtMaxLeistungMin;
END_GET
END_PROPERTY

PROPERTY p_scTable_fbrAtMinLeistung1 : CtaSysConfig.ITF_DATATYPE
GET
p_scTable_fbrAtMinLeistung1 := scParameter.scAbtauukriterium.scTable.fbrAtMinLeistung1;
END_GET
END_PROPERTY

PROPERTY p_scTable_fbrAtMinLeistung2 : CtaSysConfig.ITF_DATATYPE
GET
p_scTable_fbrAtMinLeistung2 := scParameter.scAbtauukriterium.scTable.fbrAtMinLeistung2;
END_GET
END_PROPERTY

PROPERTY p_scTable_fbrAtMinLeistungMax : CtaSysConfig.ITF_DATATYPE
GET
p_scTable_fbrAtMinLeistungMax := scParameter.scAbtauukriterium.scTable.fbrAtMinLeistungMax;
END_GET
END_PROPERTY

PROPERTY p_scTable_fbrAtMinLeistungMin : CtaSysConfig.ITF_DATATYPE
GET
p_scTable_fbrAtMinLeistungMin := scParameter.scAbtauukriterium.scTable.fbrAtMinLeistungMin;
END_GET
END_PROPERTY

PROPERTY p_scTable_fbrAussenaemperaturMax : CtaSysConfig.ITF_DATATYPE
GET
p_scTable_fbrAussenaemperaturMax := scParameter.scAbtauukriterium.scTable.fbrAussenaemperaturMax;
END_GET
END_PROPERTY

PROPERTY p_scTable_fbrAussentemperatur : CtaSysConfig.ITF_DATATYPE
GET
p_scTable_fbrAussentemperatur := scParameter.scAbtauukriterium.scTable.fbrAussentemperatur;
END_GET
END_PROPERTY

PROPERTY p_scTable_fbrAussentemperaturMin : CtaSysConfig.ITF_DATATYPE
GET
p_scTable_fbrAussentemperaturMin := scParameter.scAbtauukriterium.scTable.fbrAussentemperaturMin;
END_GET
END_PROPERTY

PROPERTY p_scTable_fbrLeistung1 : CtaSysConfig.ITF_DATATYPE
GET
p_scTable_fbrLeistung1 := scParameter.scAbtauukriterium.scTable.fbrLeistung1;
END_GET
END_PROPERTY

PROPERTY p_scTable_fbrLeistung2 : CtaSysConfig.ITF_DATATYPE
GET
p_scTable_fbrLeistung2 := scParameter.scAbtauukriterium.scTable.fbrLeistung2;
END_GET
END_PROPERTY

PROPERTY p_scTable_fbrMaxLeistung : CtaSysConfig.ITF_DATATYPE
GET
p_scTable_fbrMaxLeistung := scParameter.scAbtauukriterium.scTable.fbrMaxLeistung;
END_GET
END_PROPERTY

PROPERTY p_scTable_fbrMinLeistung : CtaSysConfig.ITF_DATATYPE
GET
p_scTable_fbrMinLeistung := scParameter.scAbtauukriterium.scTable.fbrMinLeistung;
END_GET
END_PROPERTY

PROPERTY p_scAussentemperatur_fbtAverageTimeRange : CtaSysConfig.ITF_DATATYPE
GET
p_scAussentemperatur_fbtAverageTimeRange := scParameter.scAussentemperatur.fbtAverageTimeRange;
END_GET
END_PROPERTY

PROPERTY p_scAussentemperatur_fbxAtGemittelt : CtaSysConfig.ITF_DATATYPE
GET
p_scAussentemperatur_fbxAtGemittelt := scParameter.scAussentemperatur.fbxAtGemittelt;
END_GET
END_PROPERTY

PROPERTY p_scInfluxDb_fbxEnable : CtaSysConfig.ITF_DATATYPE
GET
p_scInfluxDb_fbxEnable := scParameter.scTrend.fbxEnable;
END_GET
END_PROPERTY

PROPERTY proITF_REPORTMANAGER : CtaAppReport.ITF_REPORTMANAGER
GET
proITF_REPORTMANAGER := fbReportManager;
END_GET
END_PROPERTY

PROPERTY prorActAussentemperatur : REAL
GET
prorActAussentemperatur := SEL(scParameter.scAussentemperatur.fbxAtGemittelt.xValue,rAussentemperatur,MIN(rAussentemperatur,rAussentemperaturGemittelt));
END_GET
END_PROPERTY

PROPERTY prorActAustrittstemperatur : REAL
GET
prorActAustrittstemperatur := rAustrittstemperatur;
END_GET
END_PROPERTY

PROPERTY prorZieltemperatur : REAL
GET
prorZieltemperatur := scParameter.scAbtauuanforderung.scAbtauungHilfsenergie.fbrTempAbtauEnde.proValue;
END_GET
END_PROPERTY

PROPERTY prorActdTAbtauukriterium : REAL
GET
prorActdTAbtauukriterium := rAct_dT_Abtauukriterium;
END_GET
END_PROPERTY

PROPERTY prorAbtaukriteriumFix : REAL
GET
prorAbtaukriteriumFix := scParameter.scAbtauukriterium.fbrAbtauukriteriumFix.rValue;
END_GET
END_PROPERTY

PROPERTY prorKorrekturfaktorRk : REAL
GET
prorKorrekturfaktorRk := scParameter.scAbtauukriterium.fbrKorrekturAtLuftkühler.rValue;
END_GET
END_PROPERTY

PROPERTY prorActdTRückkühler : REAL
GET
prorActdTRückkühler := rAct_dT_Rückkühler;
END_GET
END_PROPERTY

PROPERTY prordTAuslegung : REAL
GET
prordTAuslegung := rActdTAuslegung;
END_GET
END_PROPERTY

PROPERTY prordTLeistung : REAL
GET
prordTLeistung := rActdTLeistung;
END_GET
END_PROPERTY

PROPERTY proxSperrungAktiv : BOOL
GET
proxSperrungAktiv := srSperrungAbtauung.Q1;
END_GET
END_PROPERTY

PROPERTY proudiActHilfsenergieAbtauungen : UDINT
GET
proudiActHilfsenergieAbtauungen := scParameter.scAbtauuanforderung.scAbtauungHilfsenergie.fbudiAbtauungenHiEnergie.proValue;
END_GET
END_PROPERTY

PROPERTY proudiActUmluftAbtaaungen : UDINT
GET
proudiActUmluftAbtaaungen := scParameter.scAbtauuanforderung.scUmluftabtauung.fbudiAbtauungenUmluft.proValue;
END_GET
END_PROPERTY

PROPERTY protSperrzeit : TIME
GET
protSperrzeit := TON_SperrungAbtauung.PT - TON_SperrungAbtauung.ET;
END_GET
END_PROPERTY

PROPERTY protStartverzögerung : TIME
GET
protStartverzögerung := TON_AbtauenDemand.PT - TON_AbtauenDemand.ET;
END_GET
END_PROPERTY

PROPERTY proiStatus : INT
GET
IF xDemandUmluft THEN
	proiStatus := 1;
ELSIF xDemandHilfsenergie THEN
	proiStatus := 2;
ELSIF xDemandAbtropfphase THEN
	proiStatus := 3;
ELSE
	proiStatus := 0;
END_IF
END_GET
END_PROPERTY

PROPERTY proxAcknowledge : BOOL
GET
proxAcknowledge := xAcknowledge;
END_GET
END_PROPERTY

PROPERTY proxDemandAbtauung : BOOL
GET
proxDemandAbtauung := xDemandUmluft OR xDemandHilfsenergie OR xDemandAbtropfphase;
END_GET
END_PROPERTY

PROPERTY proxDemandManualAbtauung : BOOL
GET
proxDemandManualAbtauung := (scParameter.scAbtauuanforderung.scManual.fbuiManualState.uiValue <> 0);
END_GET
END_PROPERTY

PROPERTY proxGenerelleDemand : BOOL
GET
proxGenerelleDemand := TON_AbtauenDemand.IN;
END_GET
END_PROPERTY

PROPERTY proxDemandHilfsenergie : BOOL
GET
proxDemandHilfsenergie := xDemandHilfsenergie;
END_GET
END_PROPERTY

PROPERTY proManualUmluft : BOOL
SET
IF proManualUmluft THEN
	scParameter.scAbtauuanforderung.scManual.fbuiManualState.proValue := 1;
END_IF
END_SET
GET
proManualUmluft := (scParameter.scAbtauuanforderung.scManual.fbuiManualState.proValue = 1);
END_GET
END_PROPERTY

PROPERTY proManualHilfsenergie : BOOL
SET
IF proManualHilfsenergie THEN
	scParameter.scAbtauuanforderung.scManual.fbuiManualState.proValue := 2;
END_IF
END_SET
GET
proManualHilfsenergie := (scParameter.scAbtauuanforderung.scManual.fbuiManualState.proValue = 2);
END_GET
END_PROPERTY

PROPERTY proManualBeenden : BOOL
SET
IF proManualBeenden THEN
	scParameter.scAbtauuanforderung.scManual.fbuiManualState.proValue := 3;
END_IF
END_SET
GET
proManualBeenden := (scParameter.scAbtauuanforderung.scManual.fbuiManualState.proValue = 3);
END_GET
END_PROPERTY

PROPERTY proManualQuitTime : BOOL
SET
IF proManualQuitTime THEN
	scParameter.scAbtauuanforderung.scManual.fbxManualResetLockTime.proValue := TRUE;
END_IF
END_SET
GET
proManualQuitTime := scParameter.scAbtauuanforderung.scManual.fbxManualResetLockTime.proValue;
END_GET
END_PROPERTY

PROPERTY protTimeLeftAbtropfen : TIME
GET
protTimeLeftAbtropfen := TON_Abtropfphase.PT - TON_Abtropfphase.ET;
END_GET
END_PROPERTY

PROPERTY protTimeLeftUmluft : TIME
GET
protTimeLeftUmluft := TON_AbtauungUmluft.PT - TON_AbtauungUmluft.ET;
END_GET
END_PROPERTY

PROPERTY protTimeLeftHilfsenergie : TIME
GET
protTimeLeftHilfsenergie := TON_MaxAbtauung.PT - TON_MaxAbtauung.ET;
END_GET
END_PROPERTY

PROPERTY protElapsedUmluft : TIME
GET
protElapsedUmluft := TON_AbtauungUmluft.ET;
END_GET
END_PROPERTY

PROPERTY protElapsedHilfsenergie : TIME
GET
protElapsedHilfsenergie := TON_MaxAbtauung.ET;
END_GET
END_PROPERTY

END_FUNCTION_BLOCK

// 21 Interface/ITF_Abtauung
INTERFACE ITF_Abtauung EXTENDS __SYSTEM.IQueryInterface

{attribute 'monitoring' := 'variable'}
PROPERTY proAcknowledge : BOOL
GET
END_GET
END_PROPERTY

{attribute 'monitoring' := 'variable'}
PROPERTY proAvailable : BOOL
GET
END_GET
END_PROPERTY

{attribute 'monitoring' := 'variable'}
PROPERTY proLockDown : BOOL
GET
END_GET
END_PROPERTY

PROPERTY proIsError : BOOL
GET
END_GET
END_PROPERTY

PROPERTY proIsWarning : BOOL
GET
END_GET
END_PROPERTY

PROPERTY prorActdTAbtauukriterium : REAL
GET
END_GET
END_PROPERTY

PROPERTY prorKorrekturfaktorRk : REAL
GET
END_GET
END_PROPERTY

PROPERTY prorAbtaukriteriumFix : REAL
GET
END_GET
END_PROPERTY

PROPERTY prorActAustrittstemperatur : REAL
GET
END_GET
END_PROPERTY

PROPERTY prorActAussentemperatur : REAL
GET
END_GET
END_PROPERTY

PROPERTY prorZieltemperatur : REAL
GET
END_GET
END_PROPERTY

PROPERTY proxDemandAbtauung : BOOL
GET
END_GET
END_PROPERTY

PROPERTY proxDemandManualAbtauung : BOOL
GET
END_GET
END_PROPERTY

PROPERTY proxGenerelleDemand : BOOL
GET
END_GET
END_PROPERTY

PROPERTY proxDemandHilfsenergie : BOOL
GET
END_GET
END_PROPERTY

PROPERTY proxSperrungAktiv : BOOL
GET
END_GET
END_PROPERTY

PROPERTY proudiActUmluftAbtaaungen : UDINT
GET
END_GET
END_PROPERTY

PROPERTY proudiActHilfsenergieAbtauungen : UDINT
GET
END_GET
END_PROPERTY

PROPERTY protSperrzeit : TIME
GET
END_GET
END_PROPERTY

PROPERTY protStartverzögerung : TIME
GET
END_GET
END_PROPERTY

PROPERTY proiStatus : INT
GET
END_GET
END_PROPERTY

PROPERTY proxAcknowledge : BOOL
GET
END_GET
END_PROPERTY

PROPERTY prordTAuslegung : REAL
GET
END_GET
END_PROPERTY

PROPERTY prordTLeistung : REAL
GET
END_GET
END_PROPERTY

PROPERTY prorActdTRückkühler : REAL
GET
END_GET
END_PROPERTY

PROPERTY protTimeLeftAbtropfen : TIME
GET
END_GET
END_PROPERTY

PROPERTY protTimeLeftUmluft : TIME
GET
END_GET
END_PROPERTY

PROPERTY protTimeLeftHilfsenergie : TIME
GET
END_GET
END_PROPERTY

PROPERTY protElapsedUmluft : TIME
GET
END_GET
END_PROPERTY

PROPERTY protElapsedHilfsenergie : TIME
GET
END_GET
END_PROPERTY

PROPERTY p_scAbtauungHilfsenergie_fbudiAbtauungenHiEnergie : CtaSysConfig.ITF_DATATYPE
GET
END_GET
END_PROPERTY

PROPERTY p_scAbtauungHilfsenergie_fbrTempAbtauEnde : CtaSysConfig.ITF_DATATYPE
GET
END_GET
END_PROPERTY

PROPERTY p_scAbtauungHilfsenergie_fbtMaxAbtauungHiEnergie : CtaSysConfig.ITF_DATATYPE
GET
END_GET
END_PROPERTY

PROPERTY p_scAbtauungHilfsenergie_fbiRepTilLockdown : CtaSysConfig.ITF_DATATYPE
GET
END_GET
END_PROPERTY

PROPERTY p_scAbtropfphase_fbtAbtropfzeit : CtaSysConfig.ITF_DATATYPE
GET
END_GET
END_PROPERTY

PROPERTY p_scBase_fbtAbtauverzögerung : CtaSysConfig.ITF_DATATYPE
GET
END_GET
END_PROPERTY

PROPERTY p_scBase_fbtSperrungAbtauung : CtaSysConfig.ITF_DATATYPE
GET
END_GET
END_PROPERTY

PROPERTY p_scBase_fbrAtfürAbtauusperre : CtaSysConfig.ITF_DATATYPE
GET
END_GET
END_PROPERTY

PROPERTY p_scManual_fbxManualResetLockTime : CtaSysConfig.ITF_DATATYPE
GET
END_GET
END_PROPERTY

PROPERTY p_scManual_fbuiManualState : CtaSysConfig.ITF_DATATYPE
GET
END_GET
END_PROPERTY

PROPERTY p_scUmluftabtauung_fbrTempAbtauUmluftOk : CtaSysConfig.ITF_DATATYPE
GET
END_GET
END_PROPERTY

PROPERTY p_scUmluftabtauung_fbtAbtauzeitUmluft : CtaSysConfig.ITF_DATATYPE
GET
END_GET
END_PROPERTY

PROPERTY p_scUmluftabtauung_fbudiAbtauungenUmluft : CtaSysConfig.ITF_DATATYPE
GET
END_GET
END_PROPERTY

PROPERTY p_scInfluxDb_fbxEnable : CtaSysConfig.ITF_DATATYPE
GET
END_GET
END_PROPERTY

PROPERTY p_scAbtauukriterium_fbrAbtauukriteriumFix : CtaSysConfig.ITF_DATATYPE
GET
END_GET
END_PROPERTY

PROPERTY p_scAbtauukriterium_fbrKorrekturAtLuftkühler : CtaSysConfig.ITF_DATATYPE
GET
END_GET
END_PROPERTY

PROPERTY p_scTable_fbrAtLeistungMax : CtaSysConfig.ITF_DATATYPE
GET
END_GET
END_PROPERTY

PROPERTY p_scTable_fbrAtMinLeistung1 : CtaSysConfig.ITF_DATATYPE
GET
END_GET
END_PROPERTY

PROPERTY p_scTable_fbr_dT_LeistungMin : CtaSysConfig.ITF_DATATYPE
GET
END_GET
END_PROPERTY

PROPERTY p_scTable_fbrAtMaxLeistungMax : CtaSysConfig.ITF_DATATYPE
GET
END_GET
END_PROPERTY

PROPERTY p_scTable_fbrAtMaxLeistung1 : CtaSysConfig.ITF_DATATYPE
GET
END_GET
END_PROPERTY

PROPERTY p_scTable_fbr_dT_Leistung2 : CtaSysConfig.ITF_DATATYPE
GET
END_GET
END_PROPERTY

PROPERTY p_scTable_fbr_dT_Leistung1 : CtaSysConfig.ITF_DATATYPE
GET
END_GET
END_PROPERTY

PROPERTY p_scTable_fbrAtMaxLeistung2 : CtaSysConfig.ITF_DATATYPE
GET
END_GET
END_PROPERTY

PROPERTY p_scTable_fbrAussenaemperaturMax : CtaSysConfig.ITF_DATATYPE
GET
END_GET
END_PROPERTY

PROPERTY p_scTable_fbrAussentemperaturMin : CtaSysConfig.ITF_DATATYPE
GET
END_GET
END_PROPERTY

PROPERTY p_scTable_fbrLeistung2 : CtaSysConfig.ITF_DATATYPE
GET
END_GET
END_PROPERTY

PROPERTY p_scTable_fbrMinLeistung : CtaSysConfig.ITF_DATATYPE
GET
END_GET
END_PROPERTY

PROPERTY p_scTable_fbrAtMinLeistungMax : CtaSysConfig.ITF_DATATYPE
GET
END_GET
END_PROPERTY

PROPERTY p_scTable_fbrAtLeistung1 : CtaSysConfig.ITF_DATATYPE
GET
END_GET
END_PROPERTY

PROPERTY p_scTable_fbrLeistung1 : CtaSysConfig.ITF_DATATYPE
GET
END_GET
END_PROPERTY

PROPERTY p_scTable_fbrMaxLeistung : CtaSysConfig.ITF_DATATYPE
GET
END_GET
END_PROPERTY

PROPERTY p_scTable_fbrAussentemperatur : CtaSysConfig.ITF_DATATYPE
GET
END_GET
END_PROPERTY

PROPERTY p_scTable_fbrAtMinLeistungMin : CtaSysConfig.ITF_DATATYPE
GET
END_GET
END_PROPERTY

PROPERTY p_scTable_fbrAtMinLeistung2 : CtaSysConfig.ITF_DATATYPE
GET
END_GET
END_PROPERTY

PROPERTY p_scTable_fbrAtMaxLeistungMin : CtaSysConfig.ITF_DATATYPE
GET
END_GET
END_PROPERTY

PROPERTY p_scTable_fbrAtLeistungMin : CtaSysConfig.ITF_DATATYPE
GET
END_GET
END_PROPERTY

PROPERTY p_scTable_fbrAtLeistung2 : CtaSysConfig.ITF_DATATYPE
GET
END_GET
END_PROPERTY

PROPERTY p_scTable_fbr_dT_LeistungMax : CtaSysConfig.ITF_DATATYPE
GET
END_GET
END_PROPERTY

PROPERTY p_scAussentemperatur_fbtAverageTimeRange : CtaSysConfig.ITF_DATATYPE
GET
END_GET
END_PROPERTY

PROPERTY p_scAussentemperatur_fbxAtGemittelt : CtaSysConfig.ITF_DATATYPE
GET
END_GET
END_PROPERTY

PROPERTY proConfigError : BOOL
GET
END_GET
END_PROPERTY

{attribute 'hide'} 
PROPERTY INTERNAL proITF_REPORTMANAGER : CtaAppReport.ITF_REPORTMANAGER
GET
END_GET
END_PROPERTY

PROPERTY proManualUmluft : BOOL
SET
END_SET
GET
END_GET
END_PROPERTY

PROPERTY proManualHilfsenergie : BOOL
SET
END_SET
GET
END_GET
END_PROPERTY

PROPERTY proManualBeenden : BOOL
SET
END_SET
GET
END_GET
END_PROPERTY

PROPERTY proManualQuitTime : BOOL
SET
END_SET
GET
END_GET
END_PROPERTY

END_INTERFACE

// 40 Visualizations/DIALOG/DIA_ParameterAbtauung
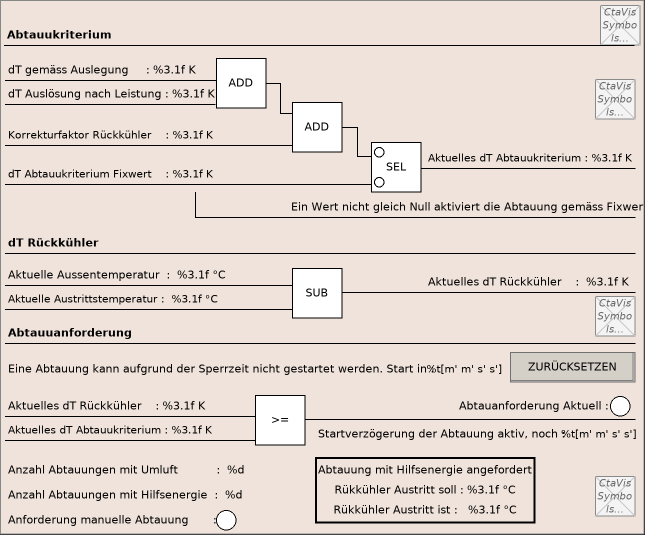
VISUALIZATION DIA_ParameterAbtauung  // 645x535
VAR_IN_OUT
	{attribute 'VAR_IN_OUT_AS_POINTER'}
	ITF_Abtauung_IN		: 	ITF_Abtauung;
END_VAR
    Rectangle (0,0 645x535)
    Image (600,5 40x40), image: CtaVisSymbols.ImagePool.close_solo_black
        OnMouseClick:  Dialog=Current Dialog, Result=OK, NumpadKeypadSet=True
    Line (5,80) (250,80)
    Line (5,104) (215,104)
    Line (5,145) (300,145)
    Line (5,184) (400,184)
    Line (250,83) (280,83)
    Rectangle (216,58 50x50), "ADD"
    Line (280,83) (280,113)
    Line (280,113) (312,113)
    Line (325,127) (357,127)
    Rectangle (292,102 50x50), "ADD"
    Label (288,197 350x20), "Ein Wert nicht gleich Null aktiviert die Abtauung gemäss Fixwert"
    Line (392,168) (635,168)
    Line (357,156) (389,156)
    Line (357,127) (357,156)
    Rectangle (371,142 50x50), "SEL"
    Ellipse (374,147 10x10), colour toggle: NOT (ITF_Abtauung_IN.prorAbtaukriteriumFix <> 0)
    Ellipse (374,177 10x10), colour toggle: (ITF_Abtauung_IN.prorAbtaukriteriumFix <> 0)
    Rectangle (5,60 210x20), "dT gemäss Auslegung : %3.1f K", text variable: ITF_Abtauung_IN.prordTAuslegung
    Rectangle (5,84 210x20), "dT Auslösung nach Leistung : %3.1f K", text variable: ITF_Abtauung_IN.prordTLeistung
    Rectangle (425,148 210x20), "Aktuelles dT Abtauukriterium : %3.1f K", text variable: ITF_Abtauung_IN.prorActdTAbtauukriterium
    Rectangle (5,125 210x20), "Korrekturfaktor Rückkühler : %3.1f K", text variable: ITF_Abtauung_IN.prorKorrekturfaktorRk
    Rectangle (5,164 210x20), "dT Abtauukriterium Fixwert : %3.1f K", text variable: ITF_Abtauung_IN.prorAbtaukriteriumFix
    Line (195,217) (635,217)
    Line (195,192) (195,217)
    Line (5,253) (635,253)
    Rectangle (5,265 220x20), "Aktuelle Aussentemperatur : %3.1f °C", text variable: ITF_Abtauung_IN.prorActAussentemperatur
    Rectangle (5,289 220x20), "Aktuelle Austrittstemperatur : %3.1f °C", text variable: ITF_Abtauung_IN.prorActAustrittstemperatur
    Rectangle (425,272 210x20), "Aktuelles dT Rückkühler : %3.1f K", text variable: ITF_Abtauung_IN.prorActdTRückkühler
    Line (5,440) (275,440)
    Line (5,416) (275,416)
    Rectangle (5,396 210x20), "Aktuelles dT Rückkühler : %3.1f K", text variable: ITF_Abtauung_IN.prorActdTRückkühler
    Rectangle (5,420 210x20), "Aktuelles dT Abtauukriterium : %3.1f K", text variable: ITF_Abtauung_IN.prorActdTAbtauukriterium
    Line (300,419) (635,419)
    Rectangle (255,395 50x50), ">="
    Label (456,396 150x20), "Abtauanforderung Aktuell :"
    Ellipse (610,396 20x20), colour toggle: ITF_Abtauung_IN.proxGenerelleDemand
    Label (315,424 240x20), "Startverzögerung der Abtauung aktiv, noch :", invisible if: NOT ITF_Abtauung_IN.proxGenerelleDemand OR NOT(ITF_Abtauung_IN.prorActdTRückkühler >= ITF_Abtauung_IN.prorActdTAbtauukriterium)
    Textfield (558,424 80x20), "%t[m' m' s' s']", text variable: ITF_Abtauung_IN.protStartverzögerung, invisible if: NOT ITF_Abtauung_IN.proxGenerelleDemand OR NOT(ITF_Abtauung_IN.prorActdTRückkühler >= ITF_Abtauung_IN.prorActdTAbtauukriterium)
    Rectangle (5,233 220x20), "dT Rückkühler"
    Rectangle (4,25 220x20), "Abtauukriterium"
    Line (4,45) (634,45)
    Rectangle (5,323 220x20), "Abtauuanforderung"
    Line (5,343) (635,343)
    Line (5,285) (300,285)
    Line (5,309) (300,309)
    Line (339,292) (635,292)
    Rectangle (292,268 50x50), "SUB"
    Image (595,79 40x40), image: CtaVisSymbols.ImagePool.gear
        OnMouseClick:  Dialog=DIA_Abtauukriterium, Parameters={ITF_Abtauung_IN: ITF_Abtauung_IN}, Selected={1: }, OpenCentered=True
    Image (595,296 40x40), image: CtaVisSymbols.ImagePool.gear
        OnMouseClick:  Dialog=DIA_Aussentemperatur, Parameters={ITF_Abtauung_IN: ITF_Abtauung_IN}, Selected={1: }, OpenCentered=True
    Label (5,359 411x20), "Eine Abtauung kann aufgrund der Sperrzeit nicht gestartet werden. Start in :", invisible if: NOT ITF_Abtauung_IN.proxSperrungAktiv
    Textfield (420,359 80x20), "%t[m' m' s' s']", text variable: ITF_Abtauung_IN.protSperrzeit, invisible if: NOT ITF_Abtauung_IN.proxSperrungAktiv
    Button (510,352 125x30), "ZURÜCKSETZEN", pressed state: ITF_Abtauung_IN.proManualQuitTime, invisible if: NOT ITF_Abtauung_IN.proxSperrungAktiv
        toggle ITF_Abtauung_IN.proManualQuitTime
        tap ITF_Abtauung_IN.proManualQuitTime
    Image (595,476 40x40), image: CtaVisSymbols.ImagePool.gear
        OnMouseClick:  Dialog=DIA_Abtauuanforderung, Parameters={ITF_Abtauung_IN: ITF_Abtauung_IN}, Selected={1: }, OpenCentered=True
    Label (5,510 250x20), "Anforderung manuelle Abtauung :"
    Ellipse (216,510 20x20), colour toggle: ITF_Abtauung_IN.proxDemandManualAbtauung
    Rectangle (5,460 250x20), "Anzahl Abtauungen mit Umluft : %d", text variable: ITF_Abtauung_IN.proudiActUmluftAbtaaungen
    Rectangle (5,485 250x20), "Anzahl Abtauungen mit Hilfsenergie : %d", text variable: ITF_Abtauung_IN.proudiActHilfsenergieAbtauungen
    Rectangle (315,460 220x20), "Abtauung mit Hilfsenergie angefordert", text variable: ITF_Abtauung_IN.proudiActUmluftAbtaaungen, invisible if: NOT ITF_Abtauung_IN.proxDemandHilfsenergie
    Rectangle (315,480 220x20), "Rükkühler Austritt soll : %3.1f °C", text variable: ITF_Abtauung_IN.prorZieltemperatur, invisible if: NOT ITF_Abtauung_IN.proxDemandHilfsenergie
    Rectangle (315,500 220x20), "Rükkühler Austritt ist : %3.1f °C", text variable: ITF_Abtauung_IN.prorActAustrittstemperatur, invisible if: NOT ITF_Abtauung_IN.proxDemandHilfsenergie
    Rectangle (315,457 220x66), invisible if: NOT ITF_Abtauung_IN.proxDemandHilfsenergie
END_VISUALIZATION

// 40 Visualizations/DIALOG/DIA_Aussentemperatur
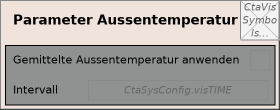
VISUALIZATION DIA_Aussentemperatur  // 280x110
VAR_IN_OUT
	{attribute 'VAR_IN_OUT_AS_POINTER'}
	ITF_Abtauung_IN	:	ITF_Abtauung;
END_VAR
    Rectangle (0,0 280x110)
    Rectangle (5,45 270x60)
    Label (10,0 350x40), "Parameter Aussentemperatur"
    Image (240,0 40x40), image: CtaVisSymbols.ImagePool.close_solo_black
        OnMouseClick:  Dialog=Current Dialog, Result=OK, NumpadKeypadSet=True
    Label (10,50 230x20), "Gemittelte Aussentemperatur anwenden"
    Frame (250,50 20x20)
        shows CtaSysConfig.visBOOL(visfbBOOLIn := ITF_Abtauung_IN.p_scAussentemperatur_fbxAtGemittelt)
    Label (10,80 60x20), "Intervall"
    Frame (88,80 180x20)
        shows CtaSysConfig.visTIME(visfbTIMEIn := ITF_Abtauung_IN.p_scAussentemperatur_fbtAverageTimeRange)
END_VISUALIZATION

// 40 Visualizations/DIALOG/DIA_Abtauukriterium
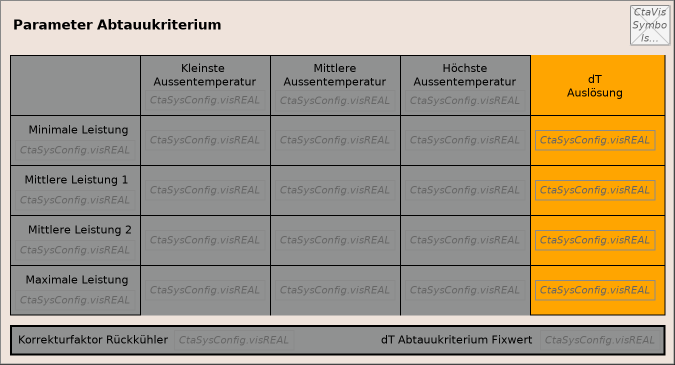
VISUALIZATION DIA_Abtauukriterium  // 675x365
VAR_IN_OUT
	{attribute 'VAR_IN_OUT_AS_POINTER'}
	ITF_Abtauung_IN	:	ITF_Abtauung;
END_VAR
    Rectangle (0,0 675x365)
    Rectangle (10,325 655x30)
    Rectangle (10,55 655x260)
    Rectangle (141,116 389x199)
    Rectangle (530,55 134x259)
    Rectangle (11,56 130x258)
    Rectangle (11,56 519x60)
    Label (10,5 350x40), "Parameter Abtauukriterium"
    Label (15,330 160x20), "Korrekturfaktor Rückkühler"
    Frame (174,330 120x20)
        shows CtaSysConfig.visREAL(visfbREALIn := ITF_Abtauung_IN.p_scAbtauukriterium_fbrKorrekturAtLuftkühler, stPhysikalischeEinheit := ' K')
    Image (630,5 40x40), image: CtaVisSymbols.ImagePool.close_solo_black
        OnMouseClick:  Dialog=Current Dialog, Result=OK, NumpadKeypadSet=True
    Frame (15,140 120x20)
        shows CtaSysConfig.visREAL(visfbREALIn := ITF_Abtauung_IN.p_scTable_fbrMinLeistung, stPhysikalischeEinheit := ' %')
    Frame (15,190 120x20)
        shows CtaSysConfig.visREAL(visfbREALIn := ITF_Abtauung_IN.p_scTable_fbrLeistung1, stPhysikalischeEinheit := ' %')
    Frame (15,240 120x20)
        shows CtaSysConfig.visREAL(visfbREALIn := ITF_Abtauung_IN.p_scTable_fbrLeistung2, stPhysikalischeEinheit := ' %')
    Frame (15,290 120x20)
        shows CtaSysConfig.visREAL(visfbREALIn := ITF_Abtauung_IN.p_scTable_fbrMaxLeistung, stPhysikalischeEinheit := ' %')
    Label (145,60 120x30), "Kleinste Aussentemperatur"
    Label (15,170 120x20), "Mittlere Leistung 1"
    Label (15,220 120x20), "Mittlere Leistung 2"
    Label (15,270 120x20), "Maximale Leistung"
    Label (275,60 120x30), "Mittlere Aussentemperatur"
    Label (405,60 120x30), "Höchste Aussentemperatur"
    Label (15,120 120x20), "Minimale Leistung"
    Frame (145,90 120x20)
        shows CtaSysConfig.visREAL(visfbREALIn := ITF_Abtauung_IN.p_scTable_fbrAussentemperaturMin, stPhysikalischeEinheit := ' °C')
    Frame (275,90 120x21)
        shows CtaSysConfig.visREAL(visfbREALIn := ITF_Abtauung_IN.p_scTable_fbrAussentemperatur, stPhysikalischeEinheit := ' °C')
    Frame (405,90 120x21)
        shows CtaSysConfig.visREAL(visfbREALIn := ITF_Abtauung_IN.p_scTable_fbrAussenaemperaturMax, stPhysikalischeEinheit := ' °C')
    Line (10,115) (665,115)
    Line (10,165) (665,165)
    Line (10,215) (665,215)
    Line (10,265) (665,265)
    Line (140,55) (140,315)
    Line (270,55) (270,315)
    Line (400,55) (400,315)
    Line (530,55) (530,315)
    Frame (145,130 120x20)
        shows CtaSysConfig.visREAL(visfbREALIn := ITF_Abtauung_IN.p_scTable_fbrAtMinLeistungMin, stPhysikalischeEinheit := ' K')
    Frame (275,130 120x20)
        shows CtaSysConfig.visREAL(visfbREALIn := ITF_Abtauung_IN.p_scTable_fbrAtLeistungMin, stPhysikalischeEinheit := ' K')
    Frame (405,130 120x20)
        shows CtaSysConfig.visREAL(visfbREALIn := ITF_Abtauung_IN.p_scTable_fbrAtMaxLeistungMin, stPhysikalischeEinheit := ' K')
    Frame (535,130 120x20)
        shows CtaSysConfig.visREAL(visfbREALIn := ITF_Abtauung_IN.p_scTable_fbr_dT_LeistungMin, stPhysikalischeEinheit := ' K')
    Frame (145,180 120x20)
        shows CtaSysConfig.visREAL(visfbREALIn := ITF_Abtauung_IN.p_scTable_fbrAtMinLeistung1, stPhysikalischeEinheit := ' K')
    Frame (275,180 120x20)
        shows CtaSysConfig.visREAL(visfbREALIn := ITF_Abtauung_IN.p_scTable_fbrAtLeistung1, stPhysikalischeEinheit := ' K')
    Frame (405,180 120x20)
        shows CtaSysConfig.visREAL(visfbREALIn := ITF_Abtauung_IN.p_scTable_fbrAtMaxLeistung1, stPhysikalischeEinheit := ' K')
    Frame (535,180 120x20)
        shows CtaSysConfig.visREAL(visfbREALIn := ITF_Abtauung_IN.p_scTable_fbr_dT_Leistung1, stPhysikalischeEinheit := ' K')
    Frame (145,230 120x20)
        shows CtaSysConfig.visREAL(visfbREALIn := ITF_Abtauung_IN.p_scTable_fbrAtMinLeistung2, stPhysikalischeEinheit := ' K')
    Frame (275,230 120x20)
        shows CtaSysConfig.visREAL(visfbREALIn := ITF_Abtauung_IN.p_scTable_fbrAtLeistung2, stPhysikalischeEinheit := ' K')
    Frame (405,230 120x20)
        shows CtaSysConfig.visREAL(visfbREALIn := ITF_Abtauung_IN.p_scTable_fbrAtMaxLeistung2, stPhysikalischeEinheit := ' K')
    Frame (535,230 120x20)
        shows CtaSysConfig.visREAL(visfbREALIn := ITF_Abtauung_IN.p_scTable_fbr_dT_Leistung2, stPhysikalischeEinheit := ' K')
    Frame (145,280 120x20)
        shows CtaSysConfig.visREAL(visfbREALIn := ITF_Abtauung_IN.p_scTable_fbrAtMinLeistungMax, stPhysikalischeEinheit := ' K')
    Frame (275,280 120x20)
        shows CtaSysConfig.visREAL(visfbREALIn := ITF_Abtauung_IN.p_scTable_fbrAtLeistungMax, stPhysikalischeEinheit := ' K')
    Frame (405,280 120x20)
        shows CtaSysConfig.visREAL(visfbREALIn := ITF_Abtauung_IN.p_scTable_fbrAtMaxLeistungMax, stPhysikalischeEinheit := ' K')
    Frame (535,280 120x20)
        shows CtaSysConfig.visREAL(visfbREALIn := ITF_Abtauung_IN.p_scTable_fbr_dT_LeistungMax, stPhysikalischeEinheit := ' K')
    Label (535,71 120x30), "dT Auslösung"
    Frame (540,330 120x20)
        shows CtaSysConfig.visREAL(visfbREALIn := ITF_Abtauung_IN.p_scAbtauukriterium_fbrAbtauukriteriumFix, stPhysikalischeEinheit := ' K')
    Label (378,330 160x20), "dT Abtauukriterium Fixwert"
END_VISUALIZATION

// 40 Visualizations/DIALOG/DIA_Abtauuanforderung
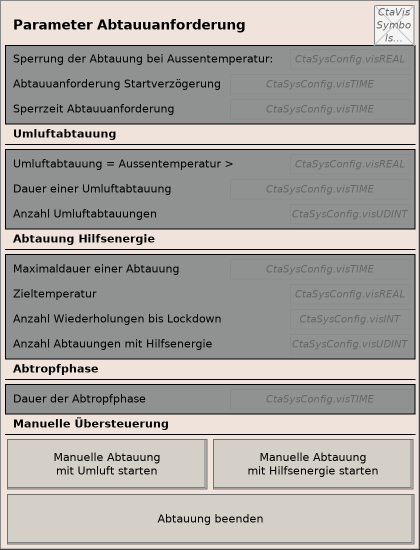
VISUALIZATION DIA_Abtauuanforderung  // 420x550
VAR_IN_OUT
	{attribute 'VAR_IN_OUT_AS_POINTER'}
	ITF_Abtauung_IN		:	ITF_Abtauung;
END_VAR
    Rectangle (0,0 420x550)
    Rectangle (5,384 410x30)
    Rectangle (5,254 410x105)
    Rectangle (5,149 410x80)
    Rectangle (5,45 410x79)
    Label (10,5 350x40), "Parameter Abtauuanforderung"
    Image (374,5 40x40), image: CtaVisSymbols.ImagePool.close_solo_black
        OnMouseClick:  Dialog=Current Dialog, Result=OK, NumpadKeypadSet=True
    Button (7,494 407x50), "Abtauung beenden", colour toggle: ITF_Abtauung_IN.proManualBeenden, pressed state: ITF_Abtauung_IN.proManualBeenden, invisible if: NOT ITF_Abtauung_IN.proxDemandAbtauung, input disabled if: ITF_Abtauung_IN.proManualBeenden
        toggle ITF_Abtauung_IN.proManualBeenden
    Label (10,74 220x20), "Abtauuanforderung Startverzögerung"
    Frame (230,74 180x20)
        shows CtaSysConfig.visTIME(visfbTIMEIn := ITF_Abtauung_IN.p_scBase_fbtAbtauverzögerung)
    Label (10,99 220x20), "Sperrzeit Abtauuanforderung"
    Frame (230,99 180x20)
        shows CtaSysConfig.visTIME(visfbTIMEIn := ITF_Abtauung_IN.p_scBase_fbtSperrungAbtauung)
    Line (5,144) (415,144)
    Rectangle (10,124 210x20), "Umluftabtauung"
    Label (10,154 220x20), "Umluftabtauung = Aussentemperatur >"
    Frame (290,154 120x20)
        shows CtaSysConfig.visREAL(visfbREALIn := ITF_Abtauung_IN.p_scUmluftabtauung_fbrTempAbtauUmluftOk, stPhysikalischeEinheit := ' °C')
    Frame (230,179 180x20)
        shows CtaSysConfig.visTIME(visfbTIMEIn := ITF_Abtauung_IN.p_scUmluftabtauung_fbtAbtauzeitUmluft)
    Label (10,179 220x20), "Dauer einer Umluftabtauung"
    Label (10,204 220x20), "Anzahl Umluftabtauungen"
    Frame (290,204 120x20)
        shows CtaSysConfig.visUDINT(visfbUDINTIn := ITF_Abtauung_IN.p_scUmluftabtauung_fbudiAbtauungenUmluft)
    Rectangle (10,229 210x20), "Abtauung Hilfsenergie"
    Line (5,249) (415,249)
    Rectangle (10,359 210x20), "Abtropfphase"
    Line (5,379) (415,379)
    Label (10,389 220x20), "Dauer der Abtropfphase"
    Frame (230,389 180x20)
        shows CtaSysConfig.visTIME(visfbTIMEIn := ITF_Abtauung_IN.p_scAbtropfphase_fbtAbtropfzeit)
    Frame (230,259 180x20)
        shows CtaSysConfig.visTIME(visfbTIMEIn := ITF_Abtauung_IN.p_scAbtauungHilfsenergie_fbtMaxAbtauungHiEnergie)
    Label (10,259 220x20), "Maximaldauer einer Abtauung"
    Label (10,334 220x20), "Anzahl Abtauungen mit Hilfsenergie"
    Label (10,309 220x20), "Anzahl Wiederholungen bis Lockdown"
    Button (7,439 200x50), "Manuelle Abtauung mit Umluft starten", colour toggle: ITF_Abtauung_IN.proManualUmluft, pressed state: ITF_Abtauung_IN.proManualUmluft, invisible if: ITF_Abtauung_IN.proxDemandAbtauung, input disabled if: ITF_Abtauung_IN.proxDemandAbtauung
        toggle ITF_Abtauung_IN.proManualUmluft
    Button (213,439 200x50), "Manuelle Abtauung mit Hilfsenergie starten", colour toggle: ITF_Abtauung_IN.proManualHilfsenergie, pressed state: ITF_Abtauung_IN.proManualHilfsenergie, invisible if: ITF_Abtauung_IN.proxDemandAbtauung, input disabled if: ITF_Abtauung_IN.proxDemandAbtauung
        toggle ITF_Abtauung_IN.proManualHilfsenergie
    Rectangle (10,414 200x20), "Manuelle Übersteuerung"
    Line (5,434) (415,434)
    Label (10,284 220x20), "Zieltemperatur"
    Frame (290,334 120x20)
        shows CtaSysConfig.visUDINT(visfbUDINTIn := ITF_Abtauung_IN.p_scAbtauungHilfsenergie_fbudiAbtauungenHiEnergie)
    Frame (290,284 120x20)
        shows CtaSysConfig.visREAL(visfbREALIn := ITF_Abtauung_IN.p_scAbtauungHilfsenergie_fbrTempAbtauEnde, stPhysikalischeEinheit := ' °C')
    Frame (290,309 120x20)
        shows CtaSysConfig.visINT(visfbINTIn := ITF_Abtauung_IN.p_scAbtauungHilfsenergie_fbiRepTilLockdown)
    Label (10,49 263x20), "Sperrung der Abtauung bei Aussentemperatur:"
    Frame (290,49 120x20)
        shows CtaSysConfig.visREAL(visfbREALIn := ITF_Abtauung_IN.p_scBase_fbrAtfürAbtauusperre, stPhysikalischeEinheit := ' °C')
END_VISUALIZATION

// 40 Visualizations/ICON/VIS_ABTAUUNG
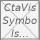
VISUALIZATION VIS_ABTAUUNG  // 40x40
VAR_INPUT
	ITF_Abtauung_IN		: 	ITF_Abtauung;
END_VAR
    Frame (0,0 40x40), invisible if: NOT( __QUERYINTERFACE(ITF_Abtauung_IN,ITF_Abtauung_IN))
        shows VIS_ABTAUUNG_CheckQuerry(ITF_Abtauung_IN := ITF_Abtauung_IN)
END_VISUALIZATION

// 40 Visualizations/ICON/VIS_ABTAUUNG_CheckQuerry
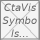
VISUALIZATION VIS_ABTAUUNG_CheckQuerry  // 40x40
VAR_INPUT
	ITF_Abtauung_IN		: 	ITF_Abtauung;
END_VAR
    Frame (0,0 40x40)
        shows VIS_ABTAUUNG_OPEN(ITF_Abtauung_IN := ITF_Abtauung_IN)
END_VISUALIZATION

// 40 Visualizations/ICON/VIS_ABTAUUNG_OPEN
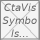
VISUALIZATION VIS_ABTAUUNG_OPEN  // 40x40
VAR_INPUT
	ITF_Abtauung_IN		: 	ITF_Abtauung;
END_VAR
    Image (0,0 40x41), invisible if: NOT __QUERYINTERFACE(ITF_Abtauung_IN,ITF_Abtauung_IN), image: CtaVisSymbols.ImagePool.snowflake_melting_icon
        OnMouseClick:  Dialog=DIA_ParameterAbtauung, Parameters={ITF_Abtauung_IN: ITF_Abtauung_IN}, Selected={0: }, OpenCentered=True
    Rectangle (0,0 40x41)
        OnMouseClick:  Dialog=DIA_ParameterAbtauung, Parameters={ITF_Abtauung_IN: ITF_Abtauung_IN}, Selected={0: }, OpenCentered=True
END_VISUALIZATION

// 40 Visualizations/VIS_AbtauungInfo
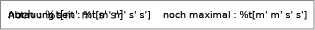
VISUALIZATION VIS_AbtauungInfo  // 315x30
VAR_INPUT
	ITF_Abtauung_IN	: ITF_Abtauung;
END_VAR
    Frame (0,0 315x30), invisible if: NOT( __QUERYINTERFACE(ITF_Abtauung_IN,ITF_Abtauung_IN))
        shows VIS_AbtauungInfoQuerry(ITF_Abtauung_IN := ITF_Abtauung_IN)
END_VISUALIZATION

// 40 Visualizations/VIS_AbtauungInfoQuerry
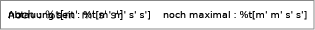
VISUALIZATION VIS_AbtauungInfoQuerry  // 315x30
VAR_INPUT
	ITF_Abtauung_IN	: ITF_Abtauung;
END_VAR
    Textfield (5,5 150x20), "Abtauung seit : %t[m' m' s' s']", text variable: ITF_Abtauung_IN.protElapsedHilfsenergie, invisible if: NOT ITF_Abtauung_IN.proxAcknowledge OR NOT(ITF_Abtauung_IN.proiStatus = 2)
    Textfield (160,5 150x20), "noch maximal : %t[m' m' s' s']", text variable: ITF_Abtauung_IN.protTimeLeftHilfsenergie, invisible if: NOT ITF_Abtauung_IN.proxAcknowledge OR NOT (ITF_Abtauung_IN.proiStatus = 2)
    Textfield (5,5 150x20), "Abtauung seit : %t[m' m' s' s']", text variable: ITF_Abtauung_IN.protElapsedUmluft, invisible if: NOT ITF_Abtauung_IN.proxAcknowledge OR NOT (ITF_Abtauung_IN.proiStatus = 1)
    Textfield (160,5 150x20), "noch maximal : %t[m' m' s' s']", text variable: ITF_Abtauung_IN.protTimeLeftUmluft, invisible if: NOT ITF_Abtauung_IN.proxAcknowledge OR NOT (ITF_Abtauung_IN.proiStatus = 1)
    Textfield (5,5 150x20), "noch : %t[m' m' s' s']", text variable: ITF_Abtauung_IN.protTimeLeftAbtropfen, invisible if: NOT ITF_Abtauung_IN.proxAcknowledge OR NOT (ITF_Abtauung_IN.proiStatus = 3)
END_VISUALIZATION

(* text list Error (id | default | de)
  0 | Keine Meldung Anstehend | Keine Meldung Anstehend
  1 | Abtauung wurde innerhalb der vorgegebenen Frist nicht erreicht | Abtauung wurde innerhalb der vorgegebenen Frist nicht erreicht
  2 | Konfigurationsfehler speichern fehlgeschlagen reboot | Konfigurationsfehler speichern fehlgeschlagen reboot
   |  |  *)

(* text list Info (id | default | de)
  0 | Keine Meldung Anstehend | Keine Meldung Anstehend
  1 | Umluftabtauung wurde gestartet | Umluftabtauung wurde gestartet
  2 | Abtauung mit Hilfsenergie wurde gestartet | Abtauung mit Hilfsenergie wurde gestartet
   |  |  *)

(* text list Warnung (id | default | de)
  3 | Keine Meldung Anstehend | Keine Meldung Anstehend
  4 | Umluftabtauung wurde gestartet | Umluftabtauung wurde gestartet
  5 | Abtauung mit Hilfsenergie wurde gestartet | Abtauung mit Hilfsenergie wurde gestartet
  6 |  | 
   |  |  *)
